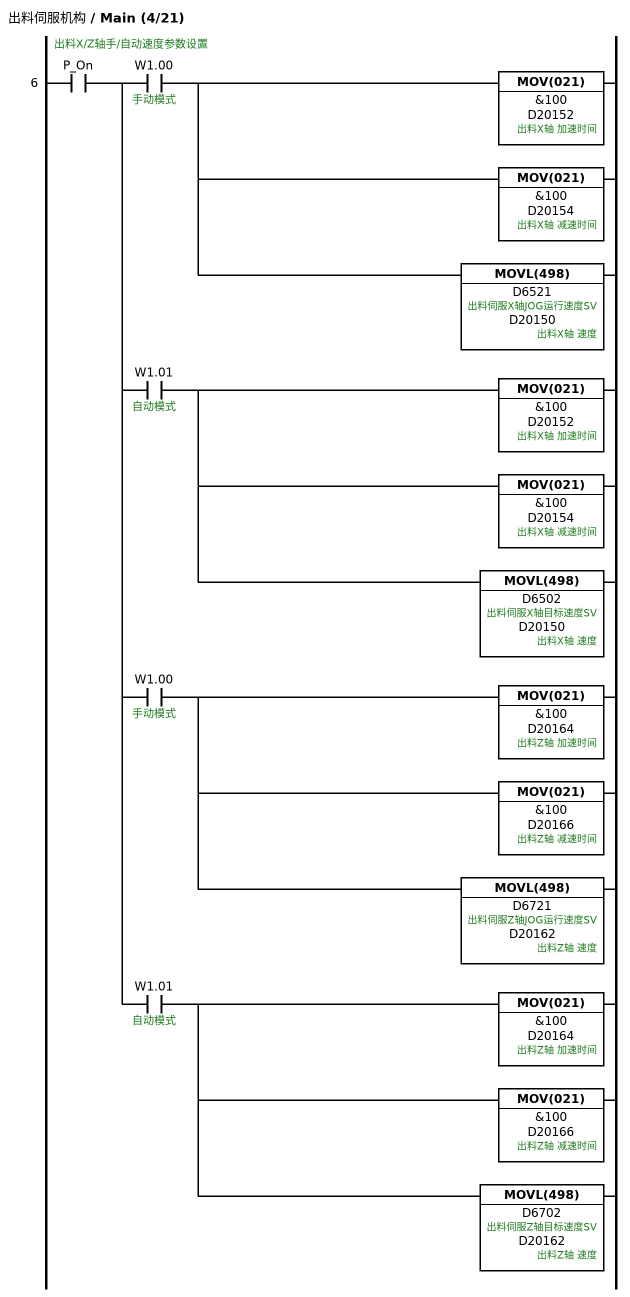
; [picture p456: 出料伺服机构 / Main, rungs 6-6]
; rung 6: 出料X/Z轴手/自动速度参数设置
LD P_On
OUT TR0
AND W1.00  ; 手动模式
MOV(021) &100 D20152  ; 出料X轴 加速时间
MOV(021) &100 D20154  ; 出料X轴 减速时间
MOVL(498) D6521 D20150  ; 出料伺服X轴JOG运行速度SV, 出料X轴 速度
LD TR0
AND W1.01  ; 自动模式
MOV(021) &100 D20152  ; 出料X轴 加速时间
MOV(021) &100 D20154  ; 出料X轴 减速时间
MOVL(498) D6502 D20150  ; 出料伺服X轴目标速度SV, 出料X轴 速度
LD TR0
AND W1.00  ; 手动模式
MOV(021) &100 D20164  ; 出料Z轴 加速时间
MOV(021) &100 D20166  ; 出料Z轴 减速时间
MOVL(498) D6721 D20162  ; 出料伺服Z轴JOG运行速度SV, 出料Z轴 速度
LD TR0
AND W1.01  ; 自动模式
MOV(021) &100 D20164  ; 出料Z轴 加速时间
MOV(021) &100 D20166  ; 出料Z轴 减速时间
MOVL(498) D6702 D20162  ; 出料伺服Z轴目标速度SV, 出料Z轴 速度

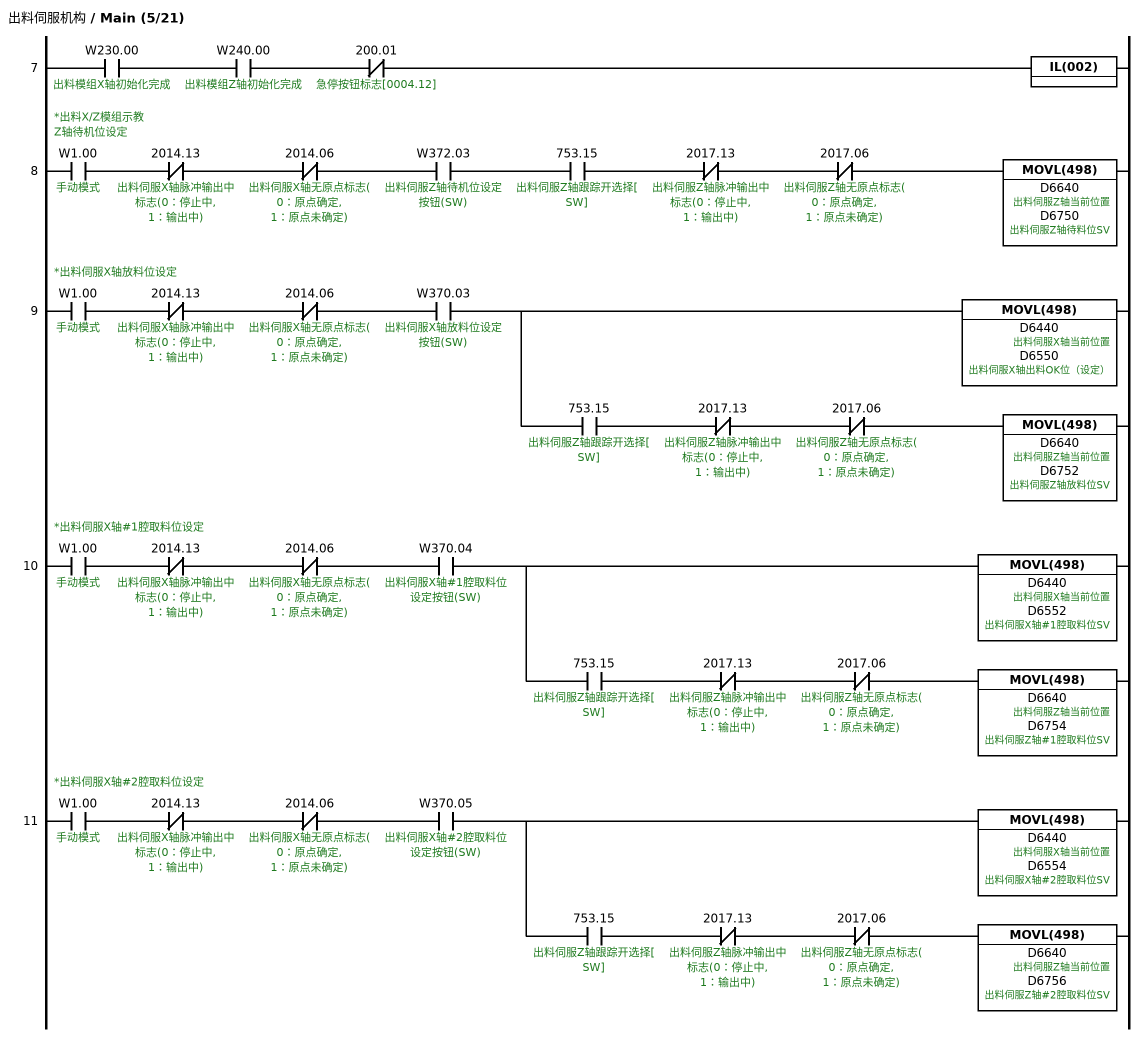
; rung 7
LD W230.00  ; 出料模组X轴初始化完成
AND W240.00  ; 出料模组Z轴初始化完成
ANDNOT 200.01  ; 急停按钮标志[0004.12]
IL(002)
; rung 8: *出料X/Z模组示教 / Z轴待机位设定
LD W1.00  ; 手动模式
ANDNOT 2014.13  ; 出料伺服X轴脉冲输出中标志(0：停止中,1：输出中)
ANDNOT 2014.06  ; 出料伺服X轴无原点标志(0：原点确定,1：原点未确定)
AND W372.03  ; 出料伺服Z轴待机位设定按钮(SW)
AND 753.15  ; 出料伺服Z轴跟踪开选择[SW]
ANDNOT 2017.13  ; 出料伺服Z轴脉冲输出中标志(0：停止中,1：输出中)
ANDNOT 2017.06  ; 出料伺服Z轴无原点标志(0：原点确定,1：原点未确定)
MOVL(498) D6640 D6750  ; 出料伺服Z轴当前位置, 出料伺服Z轴待料位SV
; rung 9: *出料伺服X轴放料位设定
LD W1.00  ; 手动模式
ANDNOT 2014.13  ; 出料伺服X轴脉冲输出中标志(0：停止中,1：输出中)
ANDNOT 2014.06  ; 出料伺服X轴无原点标志(0：原点确定,1：原点未确定)
AND W370.03  ; 出料伺服X轴放料位设定按钮(SW)
MOVL(498) D6440 D6550  ; 出料伺服X轴当前位置, 出料伺服X轴出料OK位（设定）
AND 753.15  ; 出料伺服Z轴跟踪开选择[SW]
ANDNOT 2017.13  ; 出料伺服Z轴脉冲输出中标志(0：停止中,1：输出中)
ANDNOT 2017.06  ; 出料伺服Z轴无原点标志(0：原点确定,1：原点未确定)
MOVL(498) D6640 D6752  ; 出料伺服Z轴当前位置, 出料伺服Z轴放料位SV
; rung 10: *出料伺服X轴#1腔取料位设定
LD W1.00  ; 手动模式
ANDNOT 2014.13  ; 出料伺服X轴脉冲输出中标志(0：停止中,1：输出中)
ANDNOT 2014.06  ; 出料伺服X轴无原点标志(0：原点确定,1：原点未确定)
AND W370.04  ; 出料伺服X轴#1腔取料位设定按钮(SW)
MOVL(498) D6440 D6552  ; 出料伺服X轴当前位置, 出料伺服X轴#1腔取料位SV
AND 753.15  ; 出料伺服Z轴跟踪开选择[SW]
ANDNOT 2017.13  ; 出料伺服Z轴脉冲输出中标志(0：停止中,1：输出中)
ANDNOT 2017.06  ; 出料伺服Z轴无原点标志(0：原点确定,1：原点未确定)
MOVL(498) D6640 D6754  ; 出料伺服Z轴当前位置, 出料伺服Z轴#1腔取料位SV
; rung 11: *出料伺服X轴#2腔取料位设定
LD W1.00  ; 手动模式
ANDNOT 2014.13  ; 出料伺服X轴脉冲输出中标志(0：停止中,1：输出中)
ANDNOT 2014.06  ; 出料伺服X轴无原点标志(0：原点确定,1：原点未确定)
AND W370.05  ; 出料伺服X轴#2腔取料位设定按钮(SW)
MOVL(498) D6440 D6554  ; 出料伺服X轴当前位置, 出料伺服X轴#2腔取料位SV
AND 753.15  ; 出料伺服Z轴跟踪开选择[SW]
ANDNOT 2017.13  ; 出料伺服Z轴脉冲输出中标志(0：停止中,1：输出中)
ANDNOT 2017.06  ; 出料伺服Z轴无原点标志(0：原点确定,1：原点未确定)
MOVL(498) D6640 D6756  ; 出料伺服Z轴当前位置, 出料伺服Z轴#2腔取料位SV

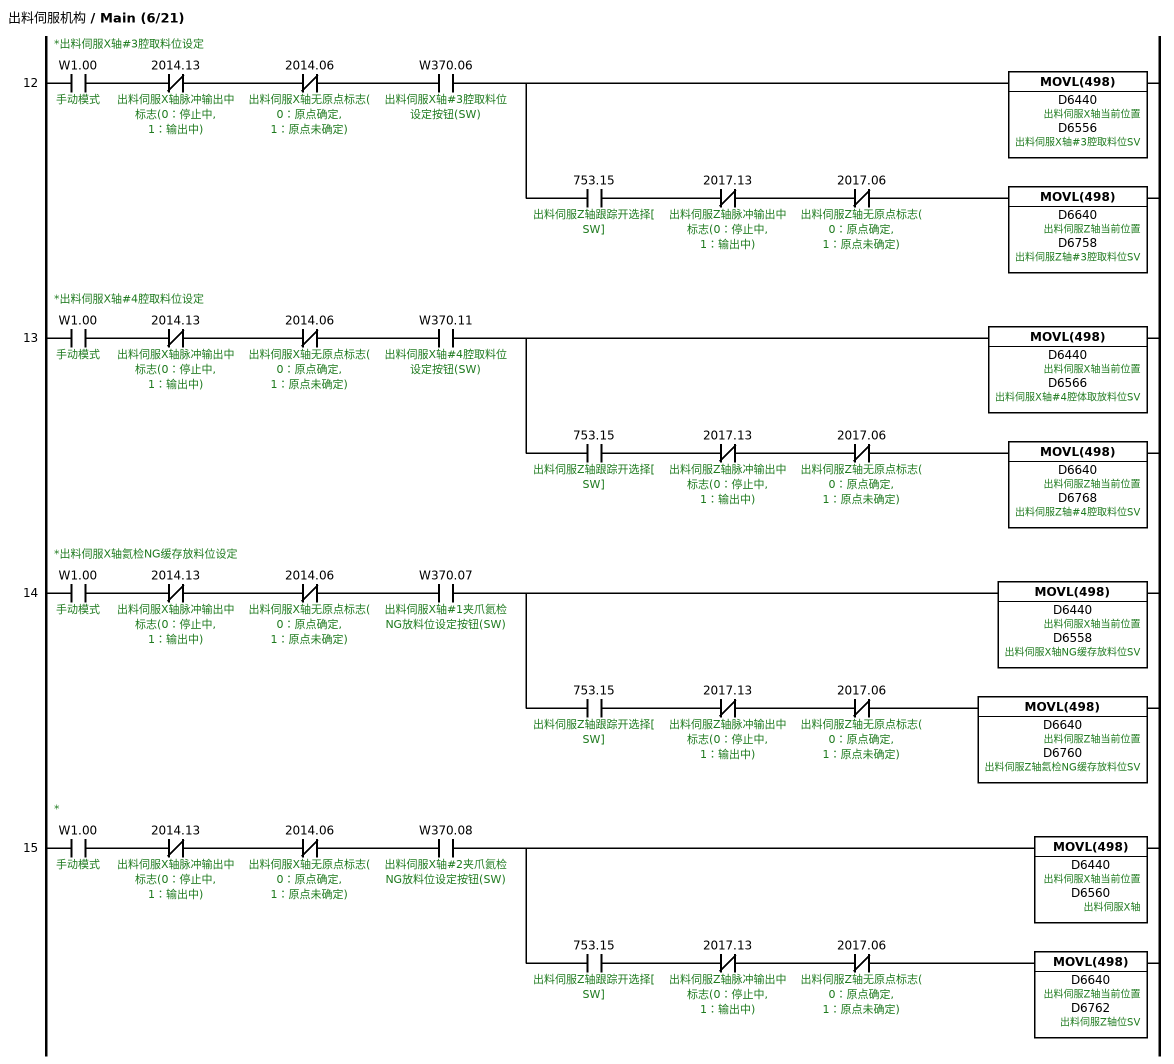
; rung 12: *出料伺服X轴#3腔取料位设定
LD W1.00  ; 手动模式
ANDNOT 2014.13  ; 出料伺服X轴脉冲输出中标志(0：停止中,1：输出中)
ANDNOT 2014.06  ; 出料伺服X轴无原点标志(0：原点确定,1：原点未确定)
AND W370.06  ; 出料伺服X轴#3腔取料位设定按钮(SW)
MOVL(498) D6440 D6556  ; 出料伺服X轴当前位置, 出料伺服X轴#3腔取料位SV
AND 753.15  ; 出料伺服Z轴跟踪开选择[SW]
ANDNOT 2017.13  ; 出料伺服Z轴脉冲输出中标志(0：停止中,1：输出中)
ANDNOT 2017.06  ; 出料伺服Z轴无原点标志(0：原点确定,1：原点未确定)
MOVL(498) D6640 D6758  ; 出料伺服Z轴当前位置, 出料伺服Z轴#3腔取料位SV
; rung 13: *出料伺服X轴#4腔取料位设定
LD W1.00  ; 手动模式
ANDNOT 2014.13  ; 出料伺服X轴脉冲输出中标志(0：停止中,1：输出中)
ANDNOT 2014.06  ; 出料伺服X轴无原点标志(0：原点确定,1：原点未确定)
AND W370.11  ; 出料伺服X轴#4腔取料位设定按钮(SW)
MOVL(498) D6440 D6566  ; 出料伺服X轴当前位置, 出料伺服X轴#4腔体取放料位SV
AND 753.15  ; 出料伺服Z轴跟踪开选择[SW]
ANDNOT 2017.13  ; 出料伺服Z轴脉冲输出中标志(0：停止中,1：输出中)
ANDNOT 2017.06  ; 出料伺服Z轴无原点标志(0：原点确定,1：原点未确定)
MOVL(498) D6640 D6768  ; 出料伺服Z轴当前位置, 出料伺服Z轴#4腔取料位SV
; rung 14: *出料伺服X轴氦检NG缓存放料位设定
LD W1.00  ; 手动模式
ANDNOT 2014.13  ; 出料伺服X轴脉冲输出中标志(0：停止中,1：输出中)
ANDNOT 2014.06  ; 出料伺服X轴无原点标志(0：原点确定,1：原点未确定)
AND W370.07  ; 出料伺服X轴#1夹爪氦检NG放料位设定按钮(SW)
MOVL(498) D6440 D6558  ; 出料伺服X轴当前位置, 出料伺服X轴NG缓存放料位SV
AND 753.15  ; 出料伺服Z轴跟踪开选择[SW]
ANDNOT 2017.13  ; 出料伺服Z轴脉冲输出中标志(0：停止中,1：输出中)
ANDNOT 2017.06  ; 出料伺服Z轴无原点标志(0：原点确定,1：原点未确定)
MOVL(498) D6640 D6760  ; 出料伺服Z轴当前位置, 出料伺服Z轴氦检NG缓存放料位SV
; rung 15: *
LD W1.00  ; 手动模式
ANDNOT 2014.13  ; 出料伺服X轴脉冲输出中标志(0：停止中,1：输出中)
ANDNOT 2014.06  ; 出料伺服X轴无原点标志(0：原点确定,1：原点未确定)
AND W370.08  ; 出料伺服X轴#2夹爪氦检NG放料位设定按钮(SW)
MOVL(498) D6440 D6560  ; 出料伺服X轴当前位置, 出料伺服X轴
AND 753.15  ; 出料伺服Z轴跟踪开选择[SW]
ANDNOT 2017.13  ; 出料伺服Z轴脉冲输出中标志(0：停止中,1：输出中)
ANDNOT 2017.06  ; 出料伺服Z轴无原点标志(0：原点确定,1：原点未确定)
MOVL(498) D6640 D6762  ; 出料伺服Z轴当前位置, 出料伺服Z轴位SV

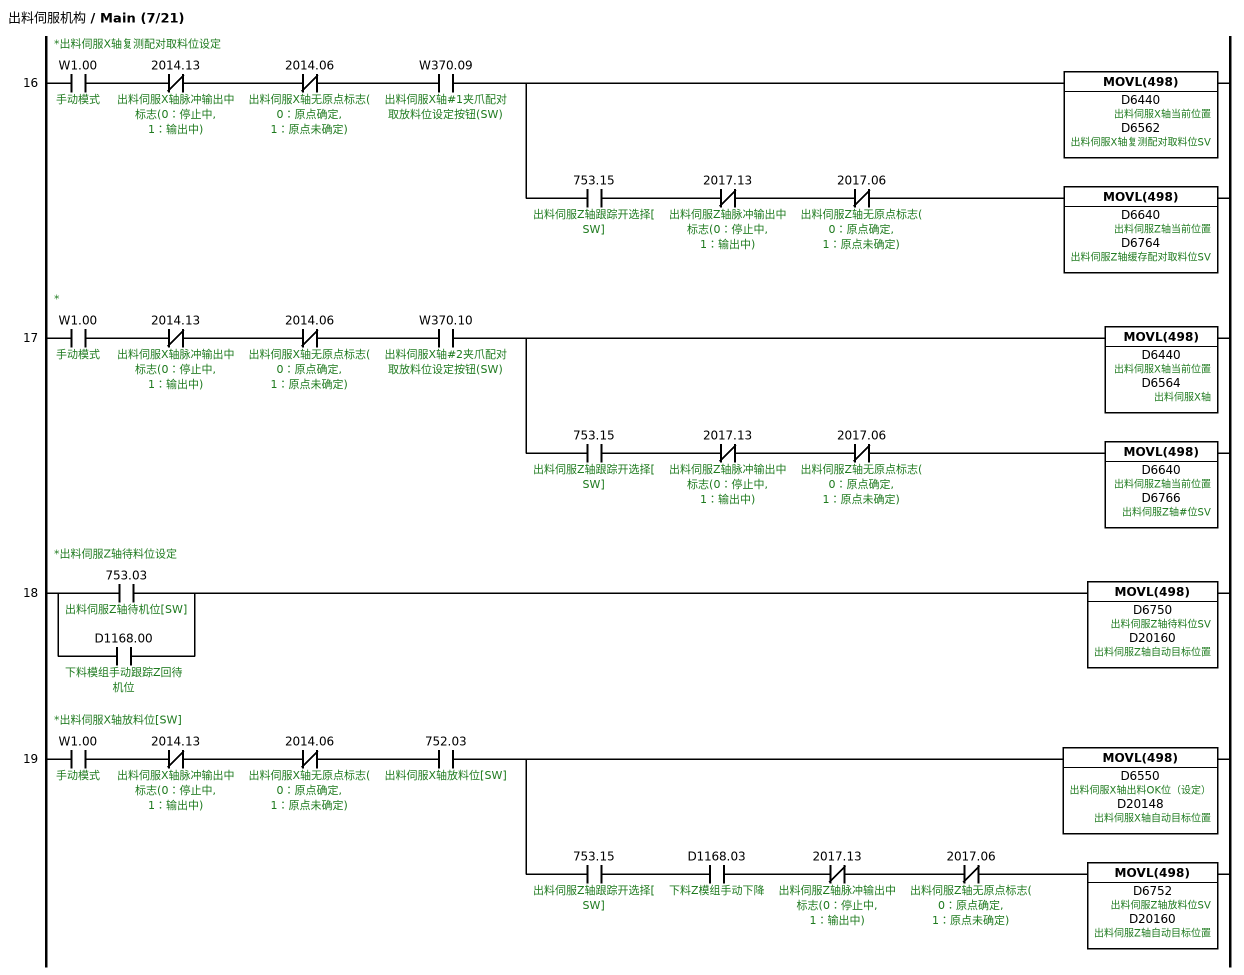
; rung 16: *出料伺服X轴复测配对取料位设定
LD W1.00  ; 手动模式
ANDNOT 2014.13  ; 出料伺服X轴脉冲输出中标志(0：停止中,1：输出中)
ANDNOT 2014.06  ; 出料伺服X轴无原点标志(0：原点确定,1：原点未确定)
AND W370.09  ; 出料伺服X轴#1夹爪配对取放料位设定按钮(SW)
MOVL(498) D6440 D6562  ; 出料伺服X轴当前位置, 出料伺服X轴复测配对取料位SV
AND 753.15  ; 出料伺服Z轴跟踪开选择[SW]
ANDNOT 2017.13  ; 出料伺服Z轴脉冲输出中标志(0：停止中,1：输出中)
ANDNOT 2017.06  ; 出料伺服Z轴无原点标志(0：原点确定,1：原点未确定)
MOVL(498) D6640 D6764  ; 出料伺服Z轴当前位置, 出料伺服Z轴缓存配对取料位SV
; rung 17: *
LD W1.00  ; 手动模式
ANDNOT 2014.13  ; 出料伺服X轴脉冲输出中标志(0：停止中,1：输出中)
ANDNOT 2014.06  ; 出料伺服X轴无原点标志(0：原点确定,1：原点未确定)
AND W370.10  ; 出料伺服X轴#2夹爪配对取放料位设定按钮(SW)
MOVL(498) D6440 D6564  ; 出料伺服X轴当前位置, 出料伺服X轴
AND 753.15  ; 出料伺服Z轴跟踪开选择[SW]
ANDNOT 2017.13  ; 出料伺服Z轴脉冲输出中标志(0：停止中,1：输出中)
ANDNOT 2017.06  ; 出料伺服Z轴无原点标志(0：原点确定,1：原点未确定)
MOVL(498) D6640 D6766  ; 出料伺服Z轴当前位置, 出料伺服Z轴#位SV
; rung 18: *出料伺服Z轴待料位设定
LD 753.03  ; 出料伺服Z轴待机位[SW]
OR D1168.00  ; 下料模组手动跟踪Z回待机位
MOVL(498) D6750 D20160  ; 出料伺服Z轴待料位SV, 出料伺服Z轴自动目标位置
; rung 19: *出料伺服X轴放料位[SW]
LD W1.00  ; 手动模式
ANDNOT 2014.13  ; 出料伺服X轴脉冲输出中标志(0：停止中,1：输出中)
ANDNOT 2014.06  ; 出料伺服X轴无原点标志(0：原点确定,1：原点未确定)
AND 752.03  ; 出料伺服X轴放料位[SW]
MOVL(498) D6550 D20148  ; 出料伺服X轴出料OK位（设定）, 出料伺服X轴自动目标位置
AND 753.15  ; 出料伺服Z轴跟踪开选择[SW]
AND D1168.03  ; 下料Z模组手动下降
ANDNOT 2017.13  ; 出料伺服Z轴脉冲输出中标志(0：停止中,1：输出中)
ANDNOT 2017.06  ; 出料伺服Z轴无原点标志(0：原点确定,1：原点未确定)
MOVL(498) D6752 D20160  ; 出料伺服Z轴放料位SV, 出料伺服Z轴自动目标位置

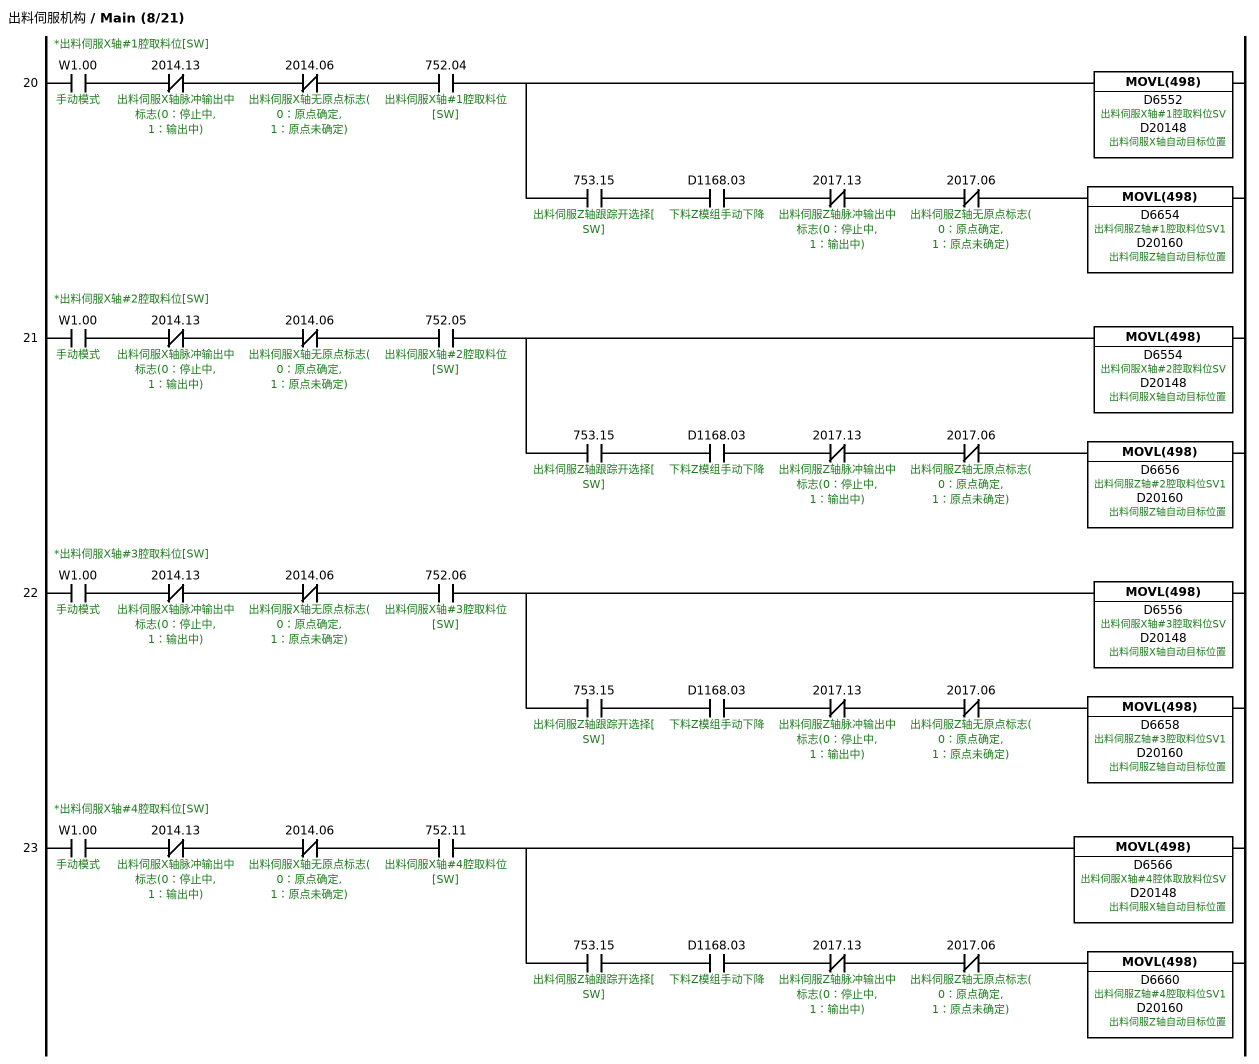
; rung 20: *出料伺服X轴#1腔取料位[SW]
LD W1.00  ; 手动模式
ANDNOT 2014.13  ; 出料伺服X轴脉冲输出中标志(0：停止中,1：输出中)
ANDNOT 2014.06  ; 出料伺服X轴无原点标志(0：原点确定,1：原点未确定)
AND 752.04  ; 出料伺服X轴#1腔取料位[SW]
MOVL(498) D6552 D20148  ; 出料伺服X轴#1腔取料位SV, 出料伺服X轴自动目标位置
AND 753.15  ; 出料伺服Z轴跟踪开选择[SW]
AND D1168.03  ; 下料Z模组手动下降
ANDNOT 2017.13  ; 出料伺服Z轴脉冲输出中标志(0：停止中,1：输出中)
ANDNOT 2017.06  ; 出料伺服Z轴无原点标志(0：原点确定,1：原点未确定)
MOVL(498) D6654 D20160  ; 出料伺服Z轴#1腔取料位SV1, 出料伺服Z轴自动目标位置
; rung 21: *出料伺服X轴#2腔取料位[SW]
LD W1.00  ; 手动模式
ANDNOT 2014.13  ; 出料伺服X轴脉冲输出中标志(0：停止中,1：输出中)
ANDNOT 2014.06  ; 出料伺服X轴无原点标志(0：原点确定,1：原点未确定)
AND 752.05  ; 出料伺服X轴#2腔取料位[SW]
MOVL(498) D6554 D20148  ; 出料伺服X轴#2腔取料位SV, 出料伺服X轴自动目标位置
AND 753.15  ; 出料伺服Z轴跟踪开选择[SW]
AND D1168.03  ; 下料Z模组手动下降
ANDNOT 2017.13  ; 出料伺服Z轴脉冲输出中标志(0：停止中,1：输出中)
ANDNOT 2017.06  ; 出料伺服Z轴无原点标志(0：原点确定,1：原点未确定)
MOVL(498) D6656 D20160  ; 出料伺服Z轴#2腔取料位SV1, 出料伺服Z轴自动目标位置
; rung 22: *出料伺服X轴#3腔取料位[SW]
LD W1.00  ; 手动模式
ANDNOT 2014.13  ; 出料伺服X轴脉冲输出中标志(0：停止中,1：输出中)
ANDNOT 2014.06  ; 出料伺服X轴无原点标志(0：原点确定,1：原点未确定)
AND 752.06  ; 出料伺服X轴#3腔取料位[SW]
MOVL(498) D6556 D20148  ; 出料伺服X轴#3腔取料位SV, 出料伺服X轴自动目标位置
AND 753.15  ; 出料伺服Z轴跟踪开选择[SW]
AND D1168.03  ; 下料Z模组手动下降
ANDNOT 2017.13  ; 出料伺服Z轴脉冲输出中标志(0：停止中,1：输出中)
ANDNOT 2017.06  ; 出料伺服Z轴无原点标志(0：原点确定,1：原点未确定)
MOVL(498) D6658 D20160  ; 出料伺服Z轴#3腔取料位SV1, 出料伺服Z轴自动目标位置
; rung 23: *出料伺服X轴#4腔取料位[SW]
LD W1.00  ; 手动模式
ANDNOT 2014.13  ; 出料伺服X轴脉冲输出中标志(0：停止中,1：输出中)
ANDNOT 2014.06  ; 出料伺服X轴无原点标志(0：原点确定,1：原点未确定)
AND 752.11  ; 出料伺服X轴#4腔取料位[SW]
MOVL(498) D6566 D20148  ; 出料伺服X轴#4腔体取放料位SV, 出料伺服X轴自动目标位置
AND 753.15  ; 出料伺服Z轴跟踪开选择[SW]
AND D1168.03  ; 下料Z模组手动下降
ANDNOT 2017.13  ; 出料伺服Z轴脉冲输出中标志(0：停止中,1：输出中)
ANDNOT 2017.06  ; 出料伺服Z轴无原点标志(0：原点确定,1：原点未确定)
MOVL(498) D6660 D20160  ; 出料伺服Z轴#4腔取料位SV1, 出料伺服Z轴自动目标位置

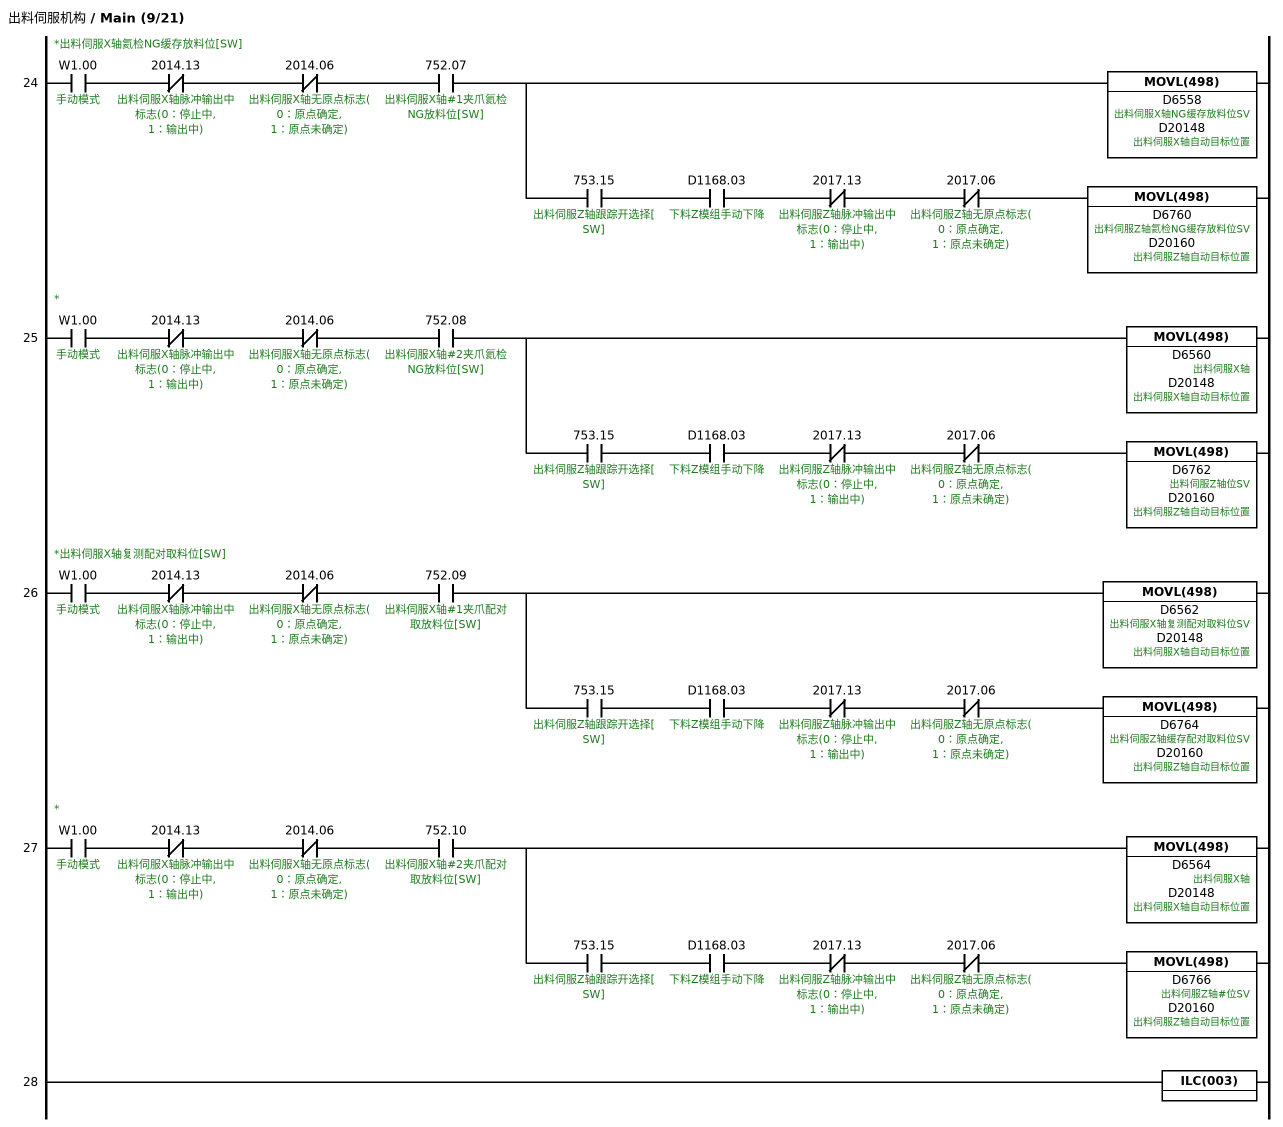
; rung 24: *出料伺服X轴氦检NG缓存放料位[SW]
LD W1.00  ; 手动模式
ANDNOT 2014.13  ; 出料伺服X轴脉冲输出中标志(0：停止中,1：输出中)
ANDNOT 2014.06  ; 出料伺服X轴无原点标志(0：原点确定,1：原点未确定)
AND 752.07  ; 出料伺服X轴#1夹爪氦检NG放料位[SW]
MOVL(498) D6558 D20148  ; 出料伺服X轴NG缓存放料位SV, 出料伺服X轴自动目标位置
AND 753.15  ; 出料伺服Z轴跟踪开选择[SW]
AND D1168.03  ; 下料Z模组手动下降
ANDNOT 2017.13  ; 出料伺服Z轴脉冲输出中标志(0：停止中,1：输出中)
ANDNOT 2017.06  ; 出料伺服Z轴无原点标志(0：原点确定,1：原点未确定)
MOVL(498) D6760 D20160  ; 出料伺服Z轴氦检NG缓存放料位SV, 出料伺服Z轴自动目标位置
; rung 25: *
LD W1.00  ; 手动模式
ANDNOT 2014.13  ; 出料伺服X轴脉冲输出中标志(0：停止中,1：输出中)
ANDNOT 2014.06  ; 出料伺服X轴无原点标志(0：原点确定,1：原点未确定)
AND 752.08  ; 出料伺服X轴#2夹爪氦检NG放料位[SW]
MOVL(498) D6560 D20148  ; 出料伺服X轴, 出料伺服X轴自动目标位置
AND 753.15  ; 出料伺服Z轴跟踪开选择[SW]
AND D1168.03  ; 下料Z模组手动下降
ANDNOT 2017.13  ; 出料伺服Z轴脉冲输出中标志(0：停止中,1：输出中)
ANDNOT 2017.06  ; 出料伺服Z轴无原点标志(0：原点确定,1：原点未确定)
MOVL(498) D6762 D20160  ; 出料伺服Z轴位SV, 出料伺服Z轴自动目标位置
; rung 26: *出料伺服X轴复测配对取料位[SW]
LD W1.00  ; 手动模式
ANDNOT 2014.13  ; 出料伺服X轴脉冲输出中标志(0：停止中,1：输出中)
ANDNOT 2014.06  ; 出料伺服X轴无原点标志(0：原点确定,1：原点未确定)
AND 752.09  ; 出料伺服X轴#1夹爪配对取放料位[SW]
MOVL(498) D6562 D20148  ; 出料伺服X轴复测配对取料位SV, 出料伺服X轴自动目标位置
AND 753.15  ; 出料伺服Z轴跟踪开选择[SW]
AND D1168.03  ; 下料Z模组手动下降
ANDNOT 2017.13  ; 出料伺服Z轴脉冲输出中标志(0：停止中,1：输出中)
ANDNOT 2017.06  ; 出料伺服Z轴无原点标志(0：原点确定,1：原点未确定)
MOVL(498) D6764 D20160  ; 出料伺服Z轴缓存配对取料位SV, 出料伺服Z轴自动目标位置
; rung 27: *
LD W1.00  ; 手动模式
ANDNOT 2014.13  ; 出料伺服X轴脉冲输出中标志(0：停止中,1：输出中)
ANDNOT 2014.06  ; 出料伺服X轴无原点标志(0：原点确定,1：原点未确定)
AND 752.10  ; 出料伺服X轴#2夹爪配对取放料位[SW]
MOVL(498) D6564 D20148  ; 出料伺服X轴, 出料伺服X轴自动目标位置
AND 753.15  ; 出料伺服Z轴跟踪开选择[SW]
AND D1168.03  ; 下料Z模组手动下降
ANDNOT 2017.13  ; 出料伺服Z轴脉冲输出中标志(0：停止中,1：输出中)
ANDNOT 2017.06  ; 出料伺服Z轴无原点标志(0：原点确定,1：原点未确定)
MOVL(498) D6766 D20160  ; 出料伺服Z轴#位SV, 出料伺服Z轴自动目标位置
; rung 28
ILC(003)

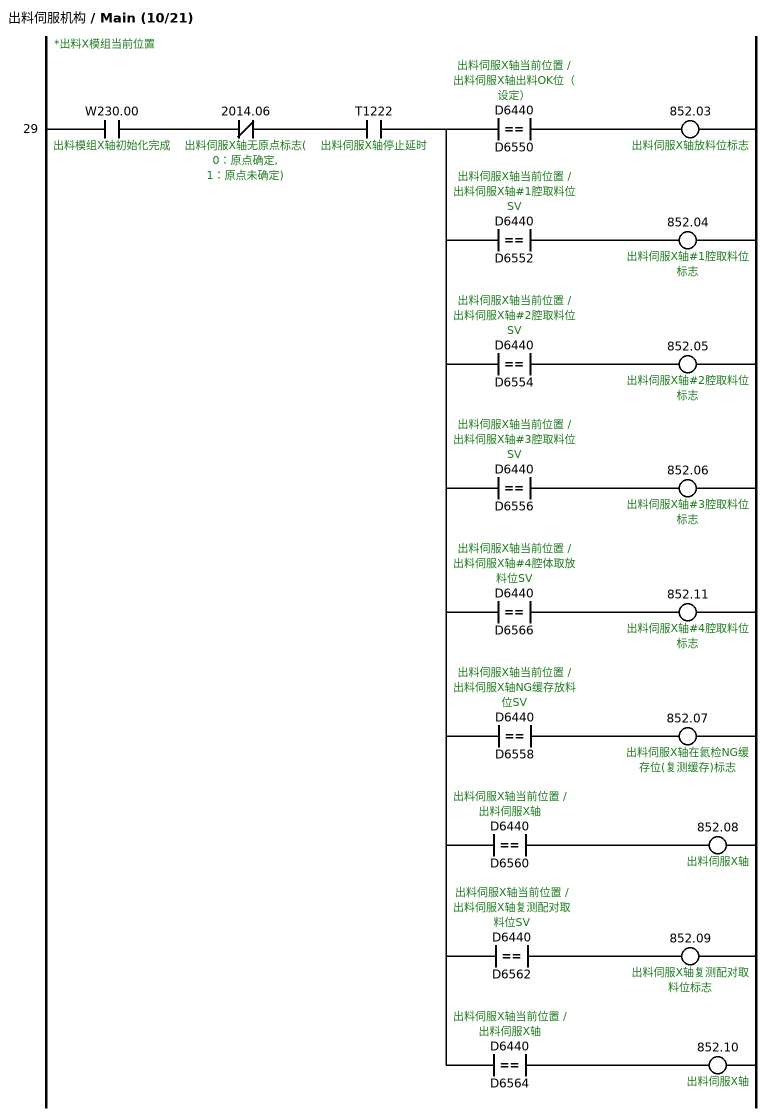
; rung 29: *出料X模组当前位置
LD W230.00  ; 出料模组X轴初始化完成
ANDNOT 2014.06  ; 出料伺服X轴无原点标志(0：原点确定,1：原点未确定)
AND T1222  ; 出料伺服X轴停止延时
OUT TR0
AND=SL(303) D6440 D6550  ; 出料伺服X轴当前位置, 出料伺服X轴出料OK位（设定）
OUT 852.03  ; 出料伺服X轴放料位标志
LD TR0
AND=SL(303) D6440 D6552  ; 出料伺服X轴当前位置, 出料伺服X轴#1腔取料位SV
OUT 852.04  ; 出料伺服X轴#1腔取料位标志
LD TR0
AND=SL(303) D6440 D6554  ; 出料伺服X轴当前位置, 出料伺服X轴#2腔取料位SV
OUT 852.05  ; 出料伺服X轴#2腔取料位标志
LD TR0
AND=SL(303) D6440 D6556  ; 出料伺服X轴当前位置, 出料伺服X轴#3腔取料位SV
OUT 852.06  ; 出料伺服X轴#3腔取料位标志
LD TR0
AND=SL(303) D6440 D6566  ; 出料伺服X轴当前位置, 出料伺服X轴#4腔体取放料位SV
OUT 852.11  ; 出料伺服X轴#4腔取料位标志
LD TR0
AND=SL(303) D6440 D6558  ; 出料伺服X轴当前位置, 出料伺服X轴NG缓存放料位SV
OUT 852.07  ; 出料伺服X轴在氦检NG缓存位(复测缓存)标志
LD TR0
AND=SL(303) D6440 D6560  ; 出料伺服X轴当前位置, 出料伺服X轴
OUT 852.08  ; 出料伺服X轴
LD TR0
AND=SL(303) D6440 D6562  ; 出料伺服X轴当前位置, 出料伺服X轴复测配对取料位SV
OUT 852.09  ; 出料伺服X轴复测配对取料位标志
LD TR0
AND=SL(303) D6440 D6564  ; 出料伺服X轴当前位置, 出料伺服X轴
OUT 852.10  ; 出料伺服X轴

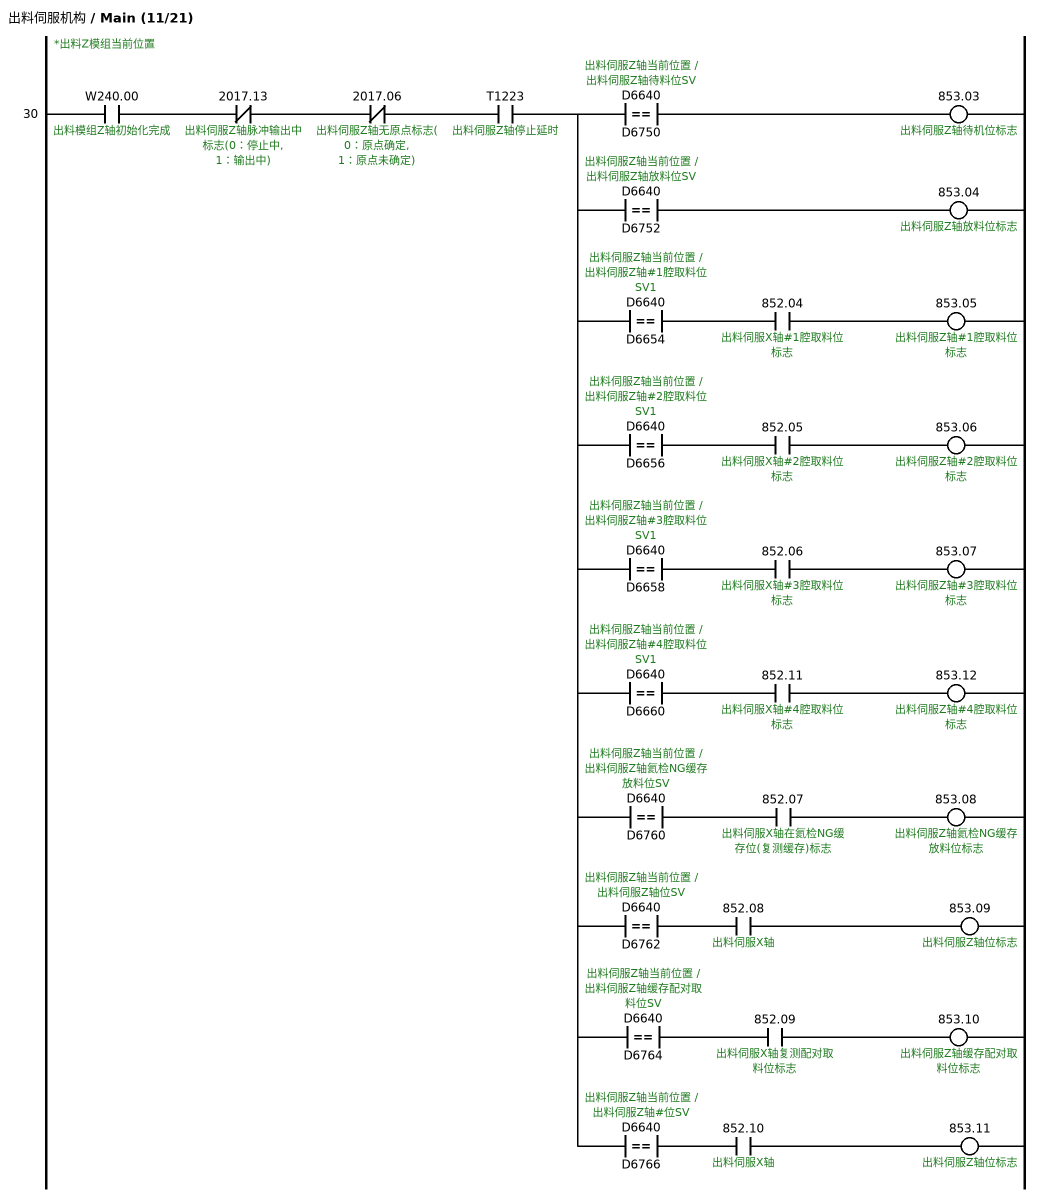
; rung 30: *出料Z模组当前位置
LD W240.00  ; 出料模组Z轴初始化完成
ANDNOT 2017.13  ; 出料伺服Z轴脉冲输出中标志(0：停止中,1：输出中)
ANDNOT 2017.06  ; 出料伺服Z轴无原点标志(0：原点确定,1：原点未确定)
AND T1223  ; 出料伺服Z轴停止延时
OUT TR0
AND=SL(303) D6640 D6750  ; 出料伺服Z轴当前位置, 出料伺服Z轴待料位SV
OUT 853.03  ; 出料伺服Z轴待机位标志
LD TR0
AND=SL(303) D6640 D6752  ; 出料伺服Z轴当前位置, 出料伺服Z轴放料位SV
OUT 853.04  ; 出料伺服Z轴放料位标志
LD TR0
AND=SL(303) D6640 D6654  ; 出料伺服Z轴当前位置, 出料伺服Z轴#1腔取料位SV1
AND 852.04  ; 出料伺服X轴#1腔取料位标志
OUT 853.05  ; 出料伺服Z轴#1腔取料位标志
LD TR0
AND=SL(303) D6640 D6656  ; 出料伺服Z轴当前位置, 出料伺服Z轴#2腔取料位SV1
AND 852.05  ; 出料伺服X轴#2腔取料位标志
OUT 853.06  ; 出料伺服Z轴#2腔取料位标志
LD TR0
AND=SL(303) D6640 D6658  ; 出料伺服Z轴当前位置, 出料伺服Z轴#3腔取料位SV1
AND 852.06  ; 出料伺服X轴#3腔取料位标志
OUT 853.07  ; 出料伺服Z轴#3腔取料位标志
LD TR0
AND=SL(303) D6640 D6660  ; 出料伺服Z轴当前位置, 出料伺服Z轴#4腔取料位SV1
AND 852.11  ; 出料伺服X轴#4腔取料位标志
OUT 853.12  ; 出料伺服Z轴#4腔取料位标志
LD TR0
AND=SL(303) D6640 D6760  ; 出料伺服Z轴当前位置, 出料伺服Z轴氦检NG缓存放料位SV
AND 852.07  ; 出料伺服X轴在氦检NG缓存位(复测缓存)标志
OUT 853.08  ; 出料伺服Z轴氦检NG缓存放料位标志
LD TR0
AND=SL(303) D6640 D6762  ; 出料伺服Z轴当前位置, 出料伺服Z轴位SV
AND 852.08  ; 出料伺服X轴
OUT 853.09  ; 出料伺服Z轴位标志
LD TR0
AND=SL(303) D6640 D6764  ; 出料伺服Z轴当前位置, 出料伺服Z轴缓存配对取料位SV
AND 852.09  ; 出料伺服X轴复测配对取料位标志
OUT 853.10  ; 出料伺服Z轴缓存配对取料位标志
LD TR0
AND=SL(303) D6640 D6766  ; 出料伺服Z轴当前位置, 出料伺服Z轴#位SV
AND 852.10  ; 出料伺服X轴
OUT 853.11  ; 出料伺服Z轴位标志

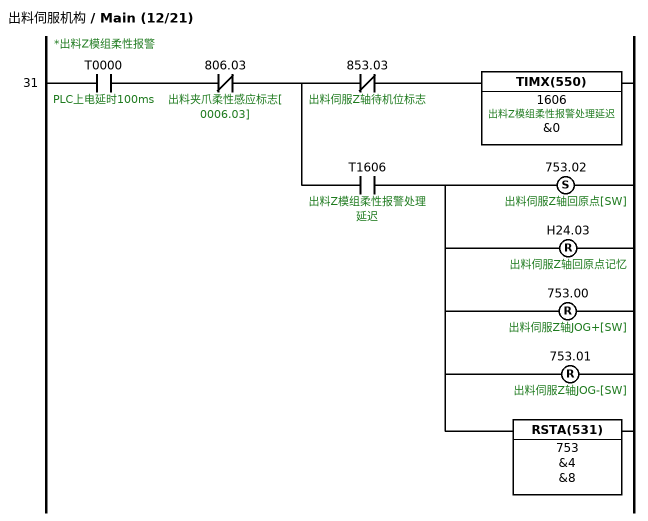
; rung 31: *出料Z模组柔性报警
LD T0000  ; PLC上电延时100ms
ANDNOT 806.03  ; 出料夹爪柔性感应标志[0006.03]
OUT TR0
ANDNOT 853.03  ; 出料伺服Z轴待机位标志
TIMX(550) 1606 &0  ; 出料Z模组柔性报警处理延迟
LD TR0
AND T1606  ; 出料Z模组柔性报警处理延迟
SET 753.02  ; 出料伺服Z轴回原点[SW]
RSET H24.03  ; 出料伺服Z轴回原点记忆
RSET 753.00  ; 出料伺服Z轴JOG+[SW]
RSET 753.01  ; 出料伺服Z轴JOG-[SW]
RSTA(531) 753 &4 &8

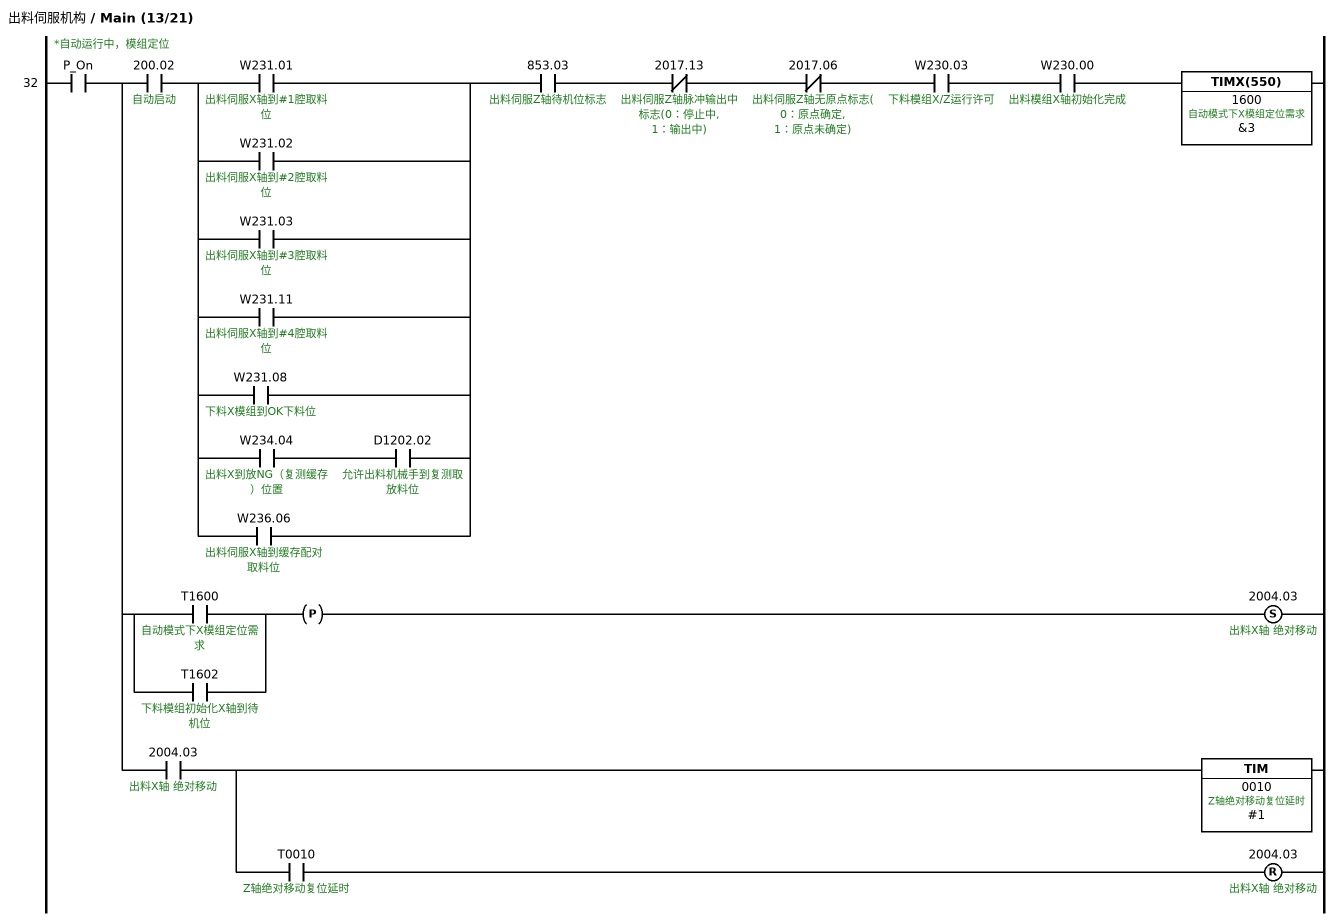
; rung 32: *自动运行中，模组定位
LD P_On
OUT TR0
AND 200.02  ; 自动启动
LD W231.01  ; 出料伺服X轴到#1腔取料位
OR W231.02  ; 出料伺服X轴到#2腔取料位
OR W231.03  ; 出料伺服X轴到#3腔取料位
OR W231.11  ; 出料伺服X轴到#4腔取料位
OR W231.08  ; 下料X模组到OK下料位
LD W234.04  ; 出料X到放NG（复测缓存）位置
AND D1202.02  ; 允许出料机械手到复测取放料位
ORLD
OR W236.06  ; 出料伺服X轴到缓存配对取料位
ANDLD
AND 853.03  ; 出料伺服Z轴待机位标志
ANDNOT 2017.13  ; 出料伺服Z轴脉冲输出中标志(0：停止中,1：输出中)
ANDNOT 2017.06  ; 出料伺服Z轴无原点标志(0：原点确定,1：原点未确定)
AND W230.03  ; 下料模组X/Z运行许可
AND W230.00  ; 出料模组X轴初始化完成
TIMX(550) 1600 &3  ; 自动模式下X模组定位需求
LD TR0
LD T1600  ; 自动模式下X模组定位需求
OR T1602  ; 下料模组初始化X轴到待机位
ANDLD
UP(521)
SET 2004.03  ; 出料X轴 绝对移动
LD TR0
AND 2004.03  ; 出料X轴 绝对移动
TIM 0010 #1  ; Z轴绝对移动复位延时
AND T0010  ; Z轴绝对移动复位延时
RSET 2004.03  ; 出料X轴 绝对移动

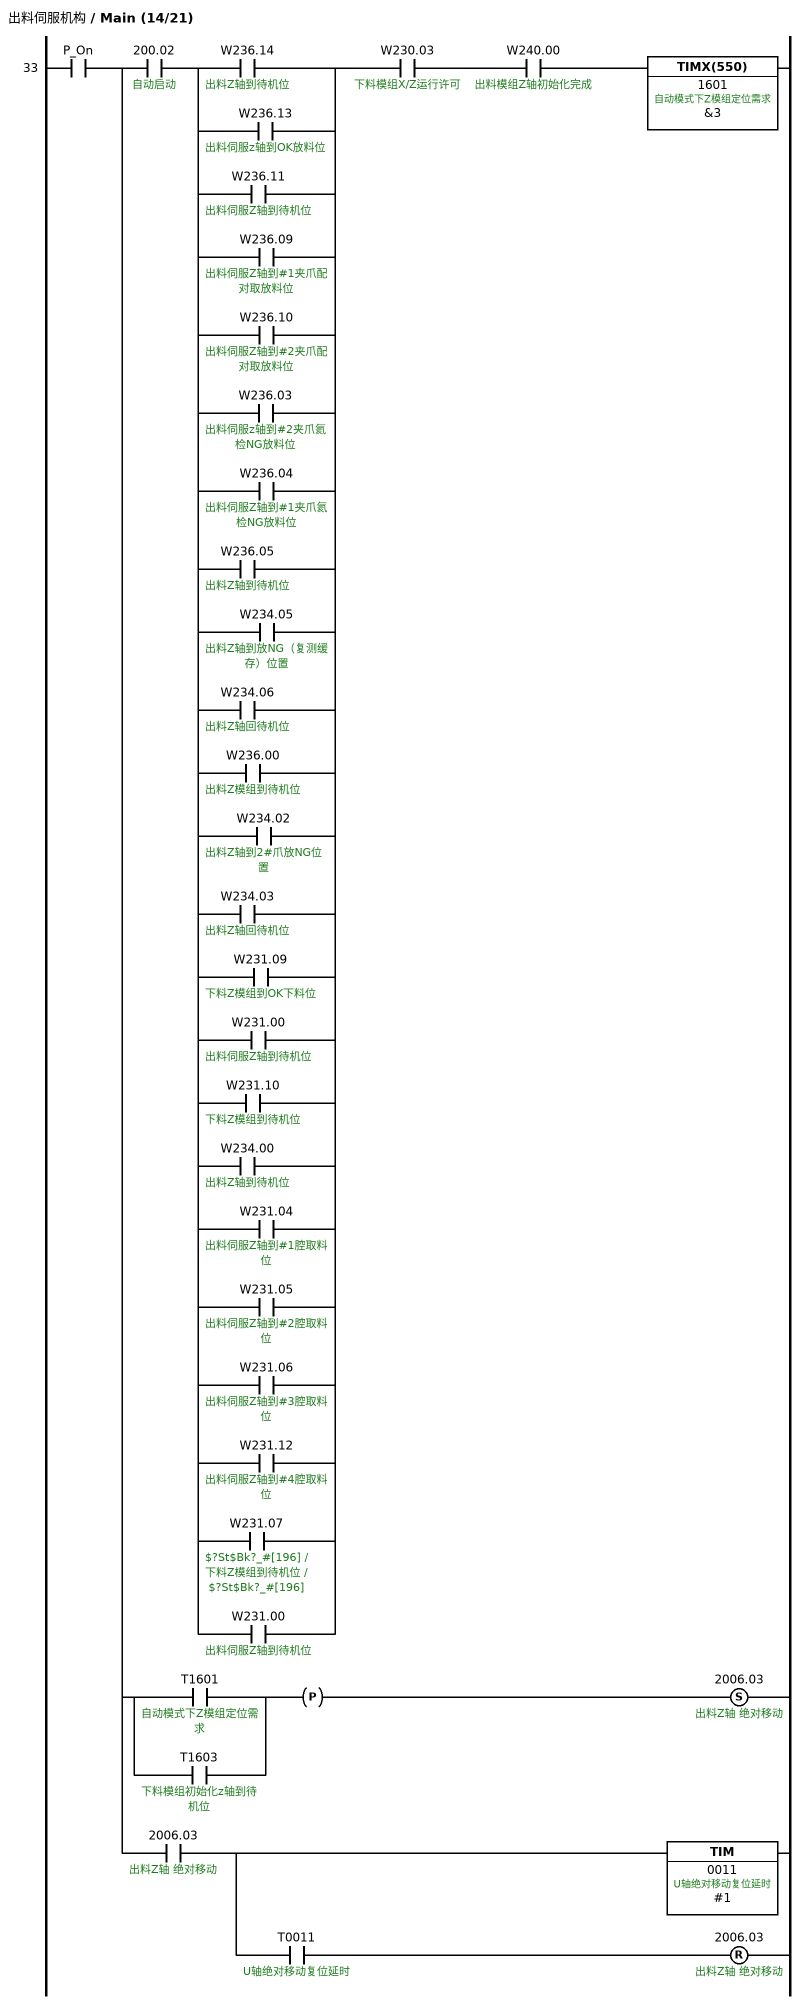
; rung 33
LD P_On
OUT TR0
AND 200.02  ; 自动启动
LD W236.14  ; 出料Z轴到待机位
OR W236.13  ; 出料伺服z轴到OK放料位
OR W236.11  ; 出料伺服Z轴到待机位
OR W236.09  ; 出料伺服Z轴到#1夹爪配对取放料位
OR W236.10  ; 出料伺服Z轴到#2夹爪配对取放料位
OR W236.03  ; 出料伺服z轴到#2夹爪氦检NG放料位
OR W236.04  ; 出料伺服Z轴到#1夹爪氦检NG放料位
OR W236.05  ; 出料Z轴到待机位
OR W234.05  ; 出料Z轴到放NG（复测缓存）位置
OR W234.06  ; 出料Z轴回待机位
OR W236.00  ; 出料Z模组到待机位
OR W234.02  ; 出料Z轴到2#爪放NG位置
OR W234.03  ; 出料Z轴回待机位
OR W231.09  ; 下料Z模组到OK下料位
OR W231.00  ; 出料伺服Z轴到待机位
OR W231.10  ; 下料Z模组到待机位
OR W234.00  ; 出料Z轴到待机位
OR W231.04  ; 出料伺服Z轴到#1腔取料位
OR W231.05  ; 出料伺服Z轴到#2腔取料位
OR W231.06  ; 出料伺服Z轴到#3腔取料位
OR W231.12  ; 出料伺服Z轴到#4腔取料位
OR W231.07  ; $?St$Bk?_#[196] / 下料Z模组到待机位 / $?St$Bk?_#[196]
OR W231.00  ; 出料伺服Z轴到待机位
ANDLD
AND W230.03  ; 下料模组X/Z运行许可
AND W240.00  ; 出料模组Z轴初始化完成
TIMX(550) 1601 &3  ; 自动模式下Z模组定位需求
LD TR0
LD T1601  ; 自动模式下Z模组定位需求
OR T1603  ; 下料模组初始化z轴到待机位
ANDLD
UP(521)
SET 2006.03  ; 出料Z轴 绝对移动
LD TR0
AND 2006.03  ; 出料Z轴 绝对移动
TIM 0011 #1  ; U轴绝对移动复位延时
AND T0011  ; U轴绝对移动复位延时
RSET 2006.03  ; 出料Z轴 绝对移动

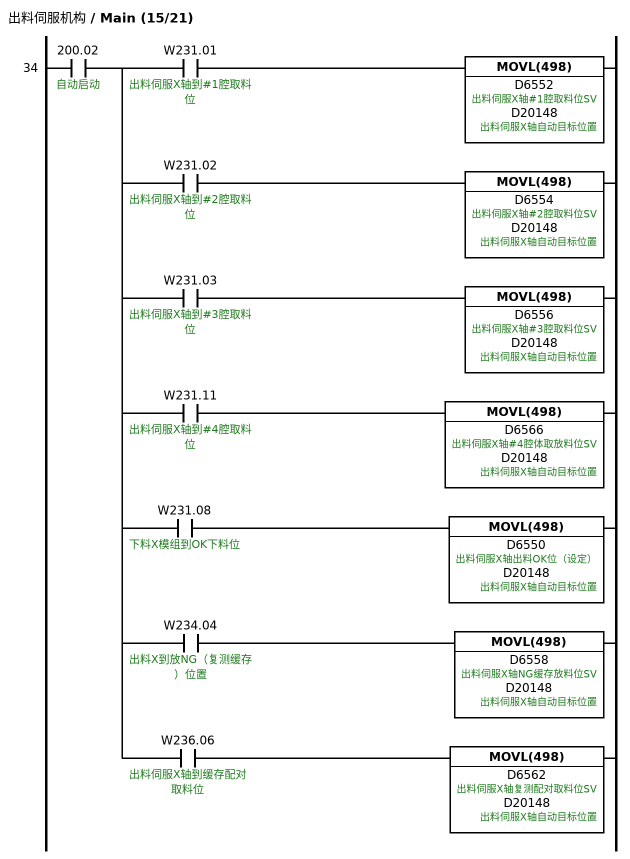
; rung 34
LD 200.02  ; 自动启动
OUT TR0
AND W231.01  ; 出料伺服X轴到#1腔取料位
MOVL(498) D6552 D20148  ; 出料伺服X轴#1腔取料位SV, 出料伺服X轴自动目标位置
LD TR0
AND W231.02  ; 出料伺服X轴到#2腔取料位
MOVL(498) D6554 D20148  ; 出料伺服X轴#2腔取料位SV, 出料伺服X轴自动目标位置
LD TR0
AND W231.03  ; 出料伺服X轴到#3腔取料位
MOVL(498) D6556 D20148  ; 出料伺服X轴#3腔取料位SV, 出料伺服X轴自动目标位置
LD TR0
AND W231.11  ; 出料伺服X轴到#4腔取料位
MOVL(498) D6566 D20148  ; 出料伺服X轴#4腔体取放料位SV, 出料伺服X轴自动目标位置
LD TR0
AND W231.08  ; 下料X模组到OK下料位
MOVL(498) D6550 D20148  ; 出料伺服X轴出料OK位（设定）, 出料伺服X轴自动目标位置
LD TR0
AND W234.04  ; 出料X到放NG（复测缓存）位置
MOVL(498) D6558 D20148  ; 出料伺服X轴NG缓存放料位SV, 出料伺服X轴自动目标位置
LD TR0
AND W236.06  ; 出料伺服X轴到缓存配对取料位
MOVL(498) D6562 D20148  ; 出料伺服X轴复测配对取料位SV, 出料伺服X轴自动目标位置

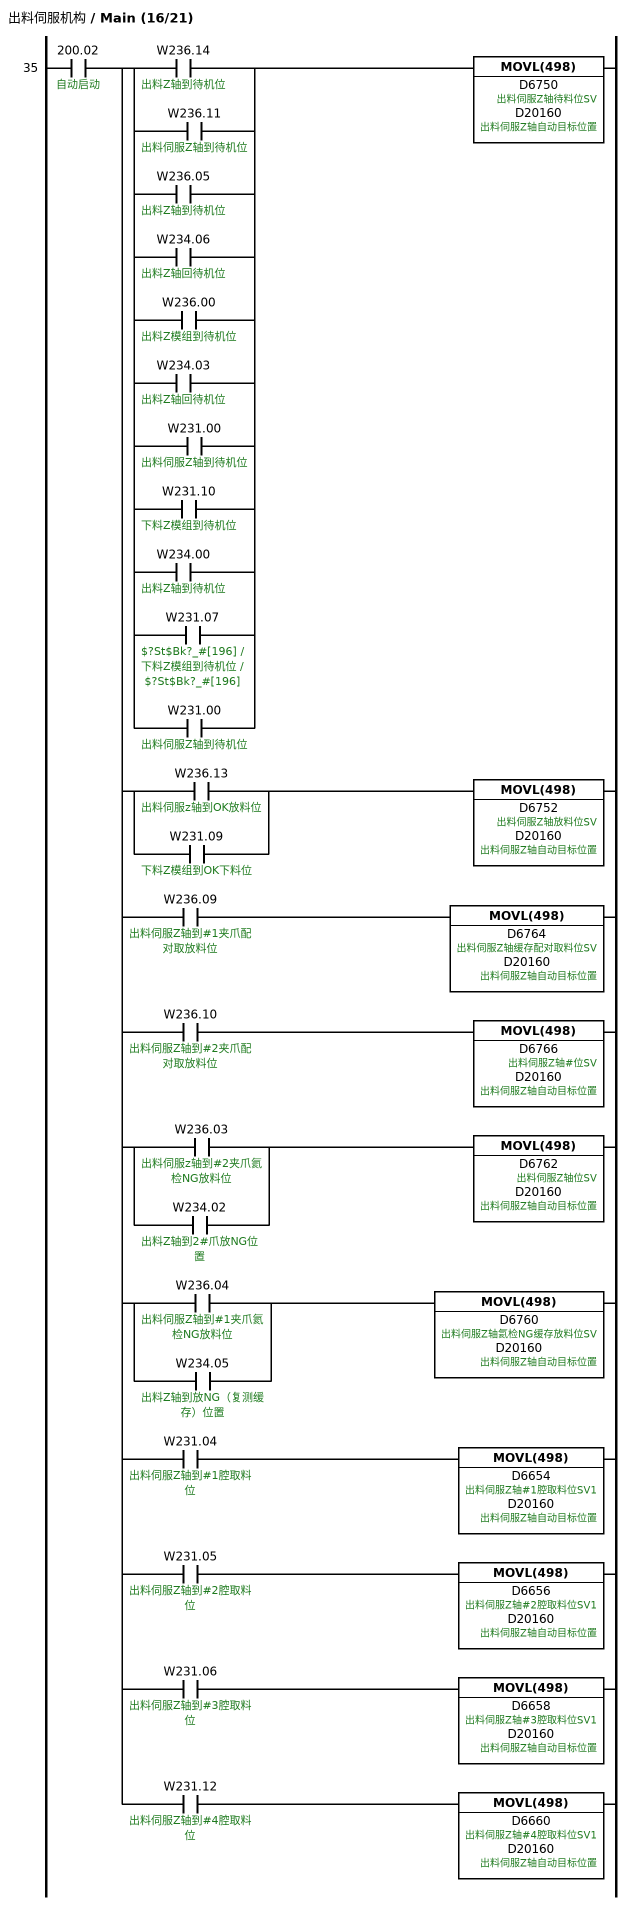
; rung 35
LD 200.02  ; 自动启动
OUT TR0
LD W236.14  ; 出料Z轴到待机位
OR W236.11  ; 出料伺服Z轴到待机位
OR W236.05  ; 出料Z轴到待机位
OR W234.06  ; 出料Z轴回待机位
OR W236.00  ; 出料Z模组到待机位
OR W234.03  ; 出料Z轴回待机位
OR W231.00  ; 出料伺服Z轴到待机位
OR W231.10  ; 下料Z模组到待机位
OR W234.00  ; 出料Z轴到待机位
OR W231.07  ; $?St$Bk?_#[196] / 下料Z模组到待机位 / $?St$Bk?_#[196]
OR W231.00  ; 出料伺服Z轴到待机位
ANDLD
MOVL(498) D6750 D20160  ; 出料伺服Z轴待料位SV, 出料伺服Z轴自动目标位置
LD TR0
LD W236.13  ; 出料伺服z轴到OK放料位
OR W231.09  ; 下料Z模组到OK下料位
ANDLD
MOVL(498) D6752 D20160  ; 出料伺服Z轴放料位SV, 出料伺服Z轴自动目标位置
LD TR0
AND W236.09  ; 出料伺服Z轴到#1夹爪配对取放料位
MOVL(498) D6764 D20160  ; 出料伺服Z轴缓存配对取料位SV, 出料伺服Z轴自动目标位置
LD TR0
AND W236.10  ; 出料伺服Z轴到#2夹爪配对取放料位
MOVL(498) D6766 D20160  ; 出料伺服Z轴#位SV, 出料伺服Z轴自动目标位置
LD TR0
LD W236.03  ; 出料伺服z轴到#2夹爪氦检NG放料位
OR W234.02  ; 出料Z轴到2#爪放NG位置
ANDLD
MOVL(498) D6762 D20160  ; 出料伺服Z轴位SV, 出料伺服Z轴自动目标位置
LD TR0
LD W236.04  ; 出料伺服Z轴到#1夹爪氦检NG放料位
OR W234.05  ; 出料Z轴到放NG（复测缓存）位置
ANDLD
MOVL(498) D6760 D20160  ; 出料伺服Z轴氦检NG缓存放料位SV, 出料伺服Z轴自动目标位置
LD TR0
AND W231.04  ; 出料伺服Z轴到#1腔取料位
MOVL(498) D6654 D20160  ; 出料伺服Z轴#1腔取料位SV1, 出料伺服Z轴自动目标位置
LD TR0
AND W231.05  ; 出料伺服Z轴到#2腔取料位
MOVL(498) D6656 D20160  ; 出料伺服Z轴#2腔取料位SV1, 出料伺服Z轴自动目标位置
LD TR0
AND W231.06  ; 出料伺服Z轴到#3腔取料位
MOVL(498) D6658 D20160  ; 出料伺服Z轴#3腔取料位SV1, 出料伺服Z轴自动目标位置
LD TR0
AND W231.12  ; 出料伺服Z轴到#4腔取料位
MOVL(498) D6660 D20160  ; 出料伺服Z轴#4腔取料位SV1, 出料伺服Z轴自动目标位置

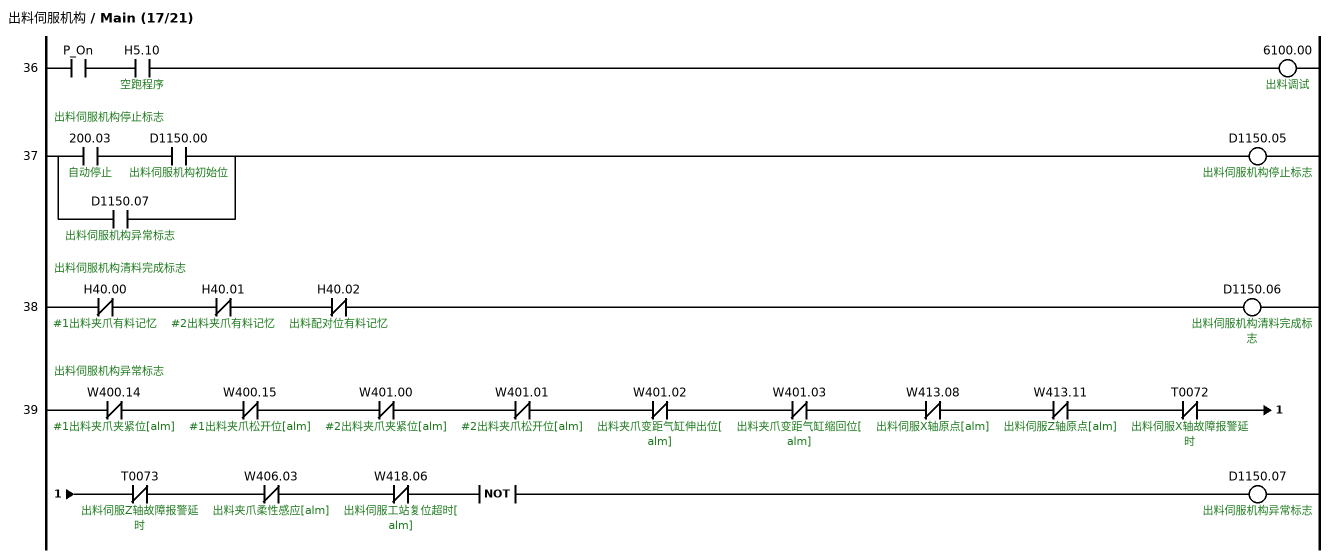
; rung 36
LD P_On
AND H5.10  ; 空跑程序
OUT 6100.00  ; 出料调试
; rung 37: 出料伺服机构停止标志
LD 200.03  ; 自动停止
AND D1150.00  ; 出料伺服机构初始位
OR D1150.07  ; 出料伺服机构异常标志
OUT D1150.05  ; 出料伺服机构停止标志
; rung 38: 出料伺服机构清料完成标志
LDNOT H40.00  ; #1出料夹爪有料记忆
ANDNOT H40.01  ; #2出料夹爪有料记忆
ANDNOT H40.02  ; 出料配对位有料记忆
OUT D1150.06  ; 出料伺服机构清料完成标志
; rung 39: 出料伺服机构异常标志
LDNOT W400.14  ; #1出料夹爪夹紧位[alm]
ANDNOT W400.15  ; #1出料夹爪松开位[alm]
ANDNOT W401.00  ; #2出料夹爪夹紧位[alm]
ANDNOT W401.01  ; #2出料夹爪松开位[alm]
ANDNOT W401.02  ; 出料夹爪变距气缸伸出位[alm]
ANDNOT W401.03  ; 出料夹爪变距气缸缩回位[alm]
ANDNOT W413.08  ; 出料伺服X轴原点[alm]
ANDNOT W413.11  ; 出料伺服Z轴原点[alm]
ANDNOT T0072  ; 出料伺服X轴故障报警延时
ANDNOT T0073  ; 出料伺服Z轴故障报警延时
ANDNOT W406.03  ; 出料夹爪柔性感应[alm]
ANDNOT W418.06  ; 出料伺服工站复位超时[alm]
NOT(520)
OUT D1150.07  ; 出料伺服机构异常标志

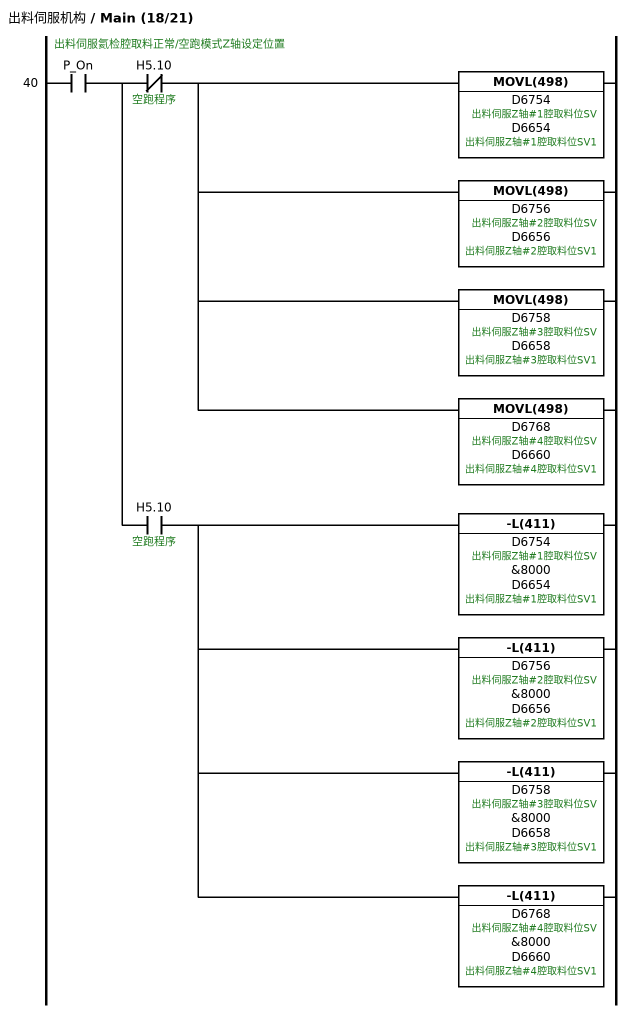
; rung 40: 出料伺服氦检腔取料正常/空跑模式Z轴设定位置
LD P_On
OUT TR0
ANDNOT H5.10  ; 空跑程序
MOVL(498) D6754 D6654  ; 出料伺服Z轴#1腔取料位SV, 出料伺服Z轴#1腔取料位SV1
MOVL(498) D6756 D6656  ; 出料伺服Z轴#2腔取料位SV, 出料伺服Z轴#2腔取料位SV1
MOVL(498) D6758 D6658  ; 出料伺服Z轴#3腔取料位SV, 出料伺服Z轴#3腔取料位SV1
MOVL(498) D6768 D6660  ; 出料伺服Z轴#4腔取料位SV, 出料伺服Z轴#4腔取料位SV1
LD TR0
AND H5.10  ; 空跑程序
-L(411) D6754 &8000 D6654  ; 出料伺服Z轴#1腔取料位SV, 出料伺服Z轴#1腔取料位SV1
-L(411) D6756 &8000 D6656  ; 出料伺服Z轴#2腔取料位SV, 出料伺服Z轴#2腔取料位SV1
-L(411) D6758 &8000 D6658  ; 出料伺服Z轴#3腔取料位SV, 出料伺服Z轴#3腔取料位SV1
-L(411) D6768 &8000 D6660  ; 出料伺服Z轴#4腔取料位SV, 出料伺服Z轴#4腔取料位SV1

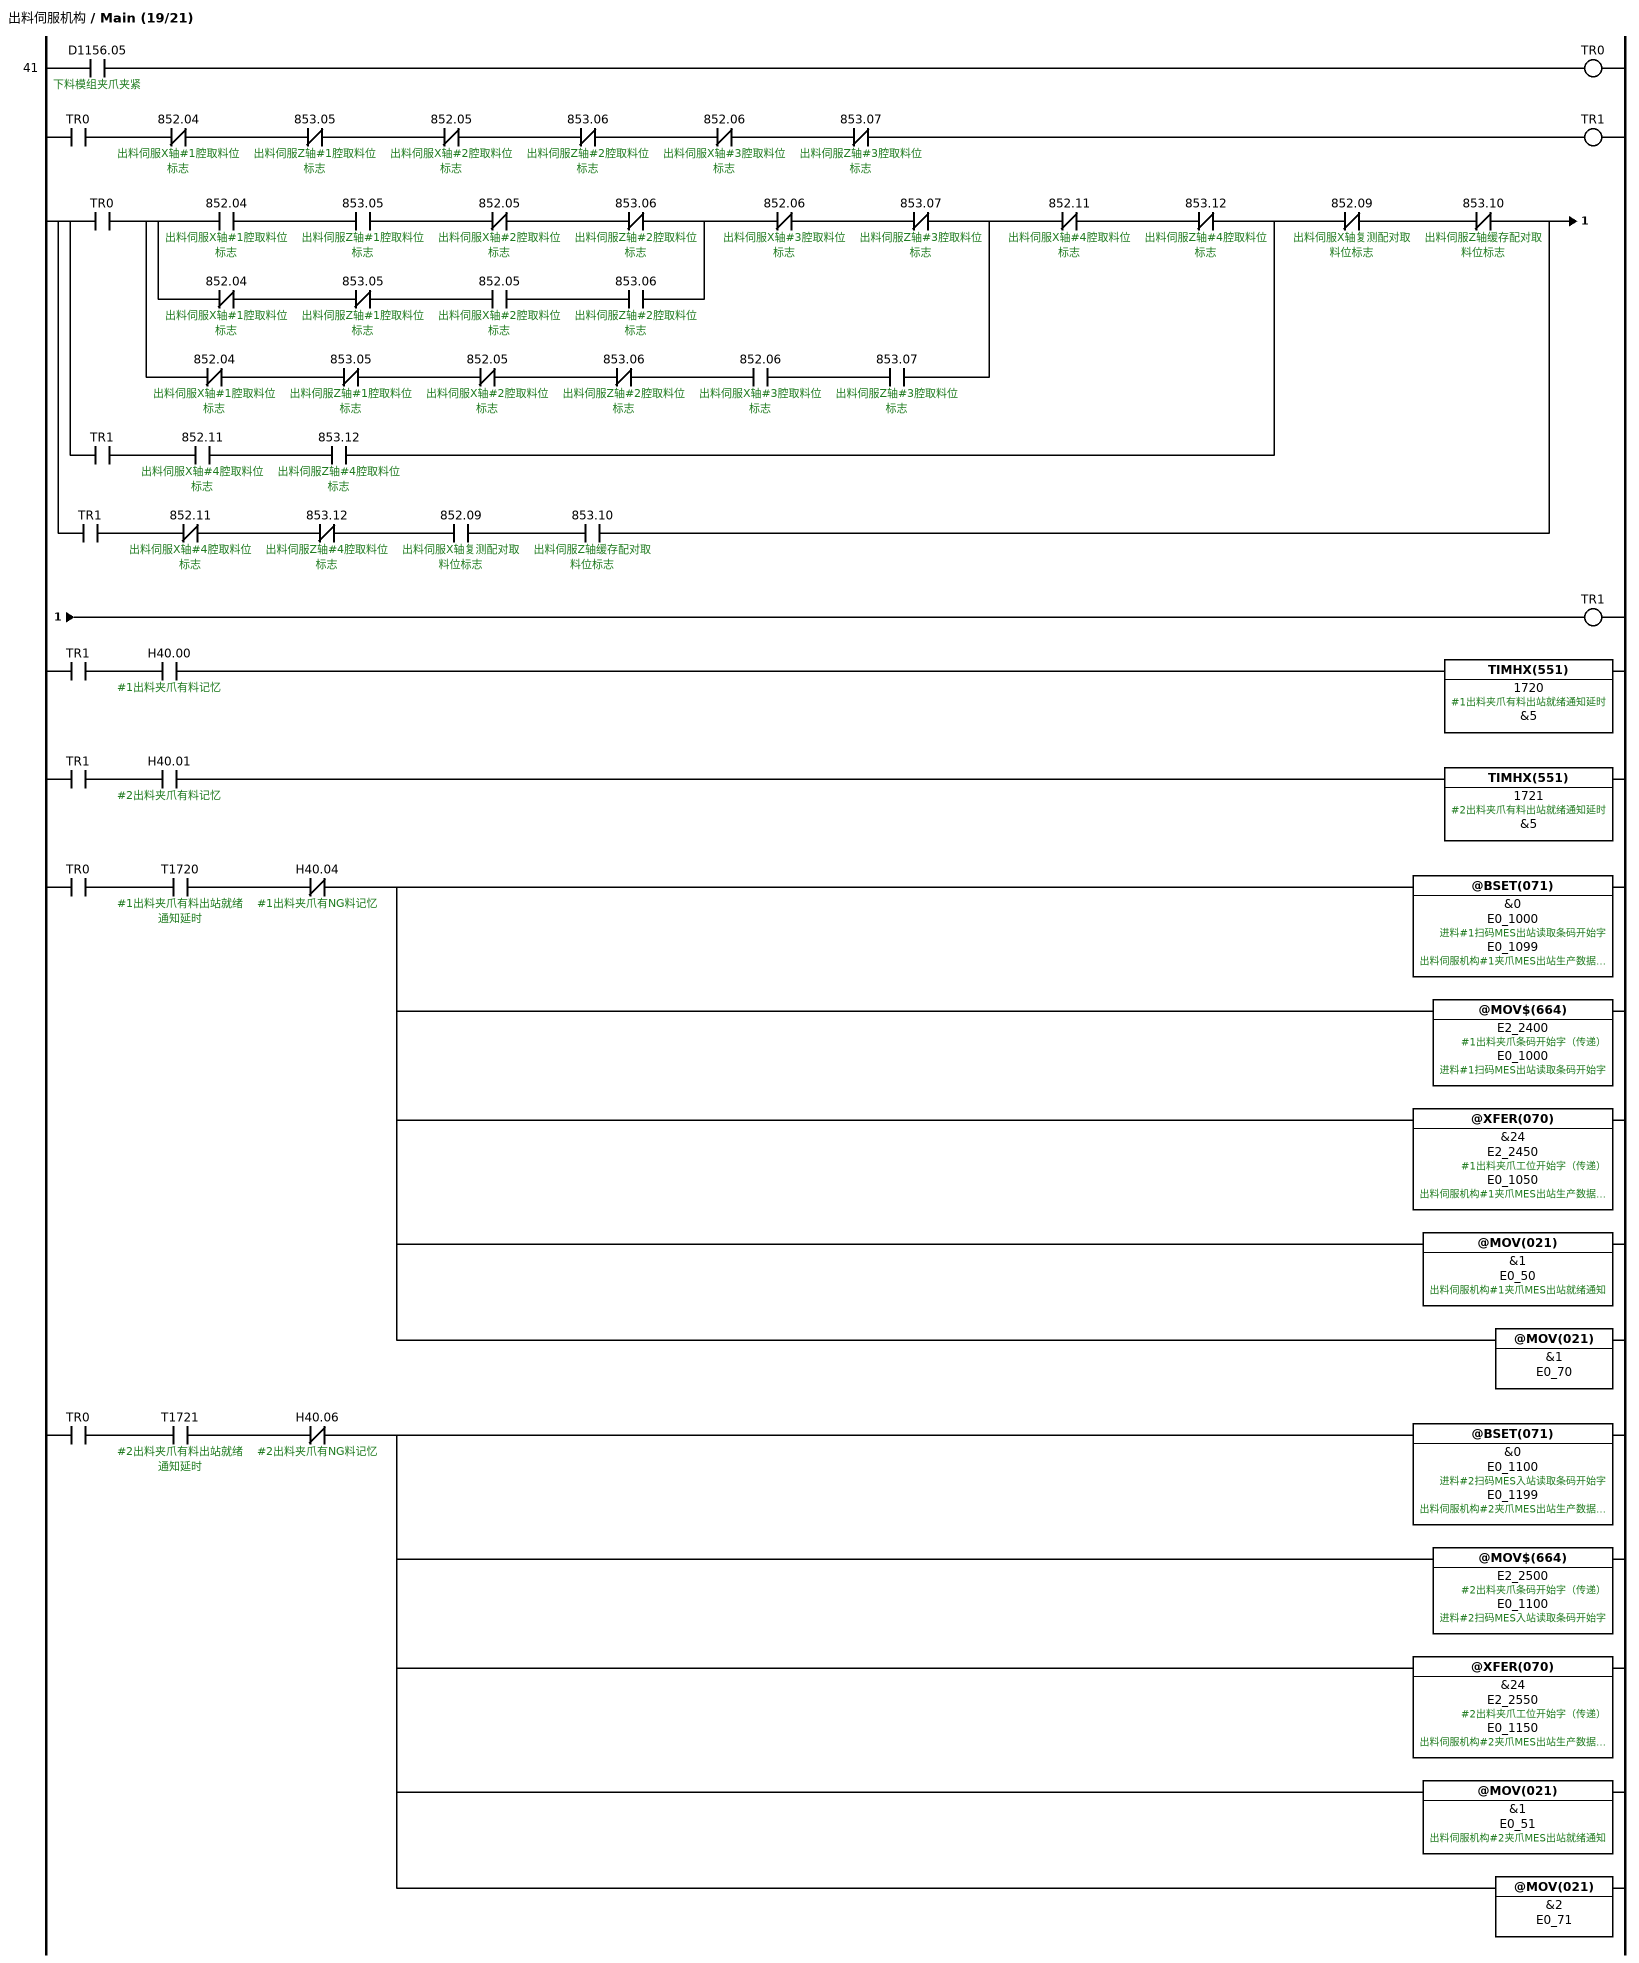
; rung 41
LD D1156.05  ; 下料模组夹爪夹紧
OUT TR0
LD 852.04  ; 出料伺服X轴#1腔取料位标志
AND 853.05  ; 出料伺服Z轴#1腔取料位标志
ANDNOT 852.05  ; 出料伺服X轴#2腔取料位标志
ANDNOT 853.06  ; 出料伺服Z轴#2腔取料位标志
LDNOT 852.04  ; 出料伺服X轴#1腔取料位标志
ANDNOT 853.05  ; 出料伺服Z轴#1腔取料位标志
AND 852.05  ; 出料伺服X轴#2腔取料位标志
AND 853.06  ; 出料伺服Z轴#2腔取料位标志
ORLD
ANDNOT 852.06  ; 出料伺服X轴#3腔取料位标志
ANDNOT 853.07  ; 出料伺服Z轴#3腔取料位标志
LDNOT 852.04  ; 出料伺服X轴#1腔取料位标志
ANDNOT 853.05  ; 出料伺服Z轴#1腔取料位标志
ANDNOT 852.05  ; 出料伺服X轴#2腔取料位标志
ANDNOT 853.06  ; 出料伺服Z轴#2腔取料位标志
AND 852.06  ; 出料伺服X轴#3腔取料位标志
AND 853.07  ; 出料伺服Z轴#3腔取料位标志
ORLD
ANDLD
ANDNOT 852.11  ; 出料伺服X轴#4腔取料位标志
ANDNOT 853.12  ; 出料伺服Z轴#4腔取料位标志
LD TR0
ANDNOT 852.04  ; 出料伺服X轴#1腔取料位标志
ANDNOT 853.05  ; 出料伺服Z轴#1腔取料位标志
ANDNOT 852.05  ; 出料伺服X轴#2腔取料位标志
ANDNOT 853.06  ; 出料伺服Z轴#2腔取料位标志
ANDNOT 852.06  ; 出料伺服X轴#3腔取料位标志
ANDNOT 853.07  ; 出料伺服Z轴#3腔取料位标志
OUT TR1
AND 852.11  ; 出料伺服X轴#4腔取料位标志
AND 853.12  ; 出料伺服Z轴#4腔取料位标志
ORLD
ANDNOT 852.09  ; 出料伺服X轴复测配对取料位标志
ANDNOT 853.10  ; 出料伺服Z轴缓存配对取料位标志
LD TR1
ANDNOT 852.11  ; 出料伺服X轴#4腔取料位标志
ANDNOT 853.12  ; 出料伺服Z轴#4腔取料位标志
AND 852.09  ; 出料伺服X轴复测配对取料位标志
AND 853.10  ; 出料伺服Z轴缓存配对取料位标志
ORLD
OUT TR1
AND H40.00  ; #1出料夹爪有料记忆
TIMHX(551) 1720 &5  ; #1出料夹爪有料出站就绪通知延时
LD TR1
AND H40.01  ; #2出料夹爪有料记忆
TIMHX(551) 1721 &5  ; #2出料夹爪有料出站就绪通知延时
LD TR0
AND T1720  ; #1出料夹爪有料出站就绪通知延时
ANDNOT H40.04  ; #1出料夹爪有NG料记忆
@BSET(071) &0 E0_1000 E0_1099  ; 进料#1扫码MES出站读取条码开始字, 出料伺服机构#1夹爪MES出站生产数据结束字
@MOV$(664) E2_2400 E0_1000  ; #1出料夹爪条码开始字（传递）, 进料#1扫码MES出站读取条码开始字
@XFER(070) &24 E2_2450 E0_1050  ; #1出料夹爪工位开始字（传递）, 出料伺服机构#1夹爪MES出站生产数据开始字
@MOV(021) &1 E0_50  ; 出料伺服机构#1夹爪MES出站就绪通知
@MOV(021) &1 E0_70
LD TR0
AND T1721  ; #2出料夹爪有料出站就绪通知延时
ANDNOT H40.06  ; #2出料夹爪有NG料记忆
@BSET(071) &0 E0_1100 E0_1199  ; 进料#2扫码MES入站读取条码开始字, 出料伺服机构#2夹爪MES出站生产数据结束字
@MOV$(664) E2_2500 E0_1100  ; #2出料夹爪条码开始字（传递）, 进料#2扫码MES入站读取条码开始字
@XFER(070) &24 E2_2550 E0_1150  ; #2出料夹爪工位开始字（传递）, 出料伺服机构#2夹爪MES出站生产数据开始字
@MOV(021) &1 E0_51  ; 出料伺服机构#2夹爪MES出站就绪通知
@MOV(021) &2 E0_71

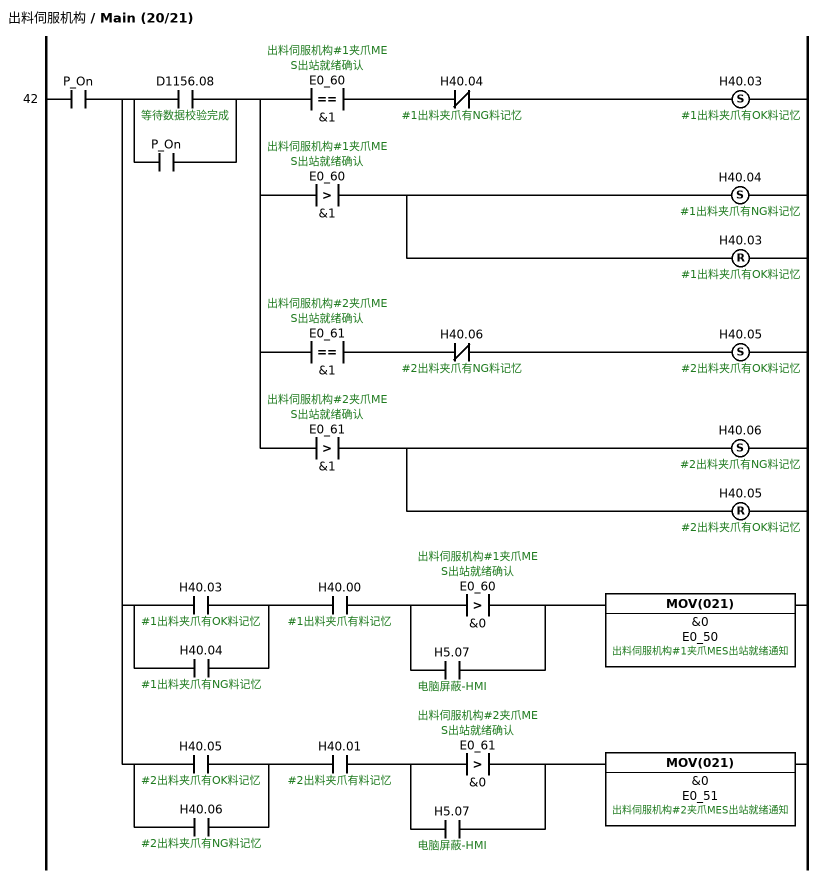
; rung 42
LD P_On
OUT TR0
LD D1156.08  ; 等待数据校验完成
OR P_On
ANDLD
OUT TR1
AND=(300) E0_60 &1  ; 出料伺服机构#1夹爪MES出站就绪确认
ANDNOT H40.04  ; #1出料夹爪有NG料记忆
SET H40.03  ; #1出料夹爪有OK料记忆
LD TR1
AND>(320) E0_60 &1  ; 出料伺服机构#1夹爪MES出站就绪确认
SET H40.04  ; #1出料夹爪有NG料记忆
RSET H40.03  ; #1出料夹爪有OK料记忆
LD TR1
AND=(300) E0_61 &1  ; 出料伺服机构#2夹爪MES出站就绪确认
ANDNOT H40.06  ; #2出料夹爪有NG料记忆
SET H40.05  ; #2出料夹爪有OK料记忆
LD TR1
AND>(320) E0_61 &1  ; 出料伺服机构#2夹爪MES出站就绪确认
SET H40.06  ; #2出料夹爪有NG料记忆
RSET H40.05  ; #2出料夹爪有OK料记忆
LD TR0
LD H40.03  ; #1出料夹爪有OK料记忆
OR H40.04  ; #1出料夹爪有NG料记忆
ANDLD
AND H40.00  ; #1出料夹爪有料记忆
LD>(320) E0_60 &0  ; 出料伺服机构#1夹爪MES出站就绪确认
OR H5.07  ; 电脑屏蔽-HMI
ANDLD
MOV(021) &0 E0_50  ; 出料伺服机构#1夹爪MES出站就绪通知
LD TR0
LD H40.05  ; #2出料夹爪有OK料记忆
OR H40.06  ; #2出料夹爪有NG料记忆
ANDLD
AND H40.01  ; #2出料夹爪有料记忆
LD>(320) E0_61 &0  ; 出料伺服机构#2夹爪MES出站就绪确认
OR H5.07  ; 电脑屏蔽-HMI
ANDLD
MOV(021) &0 E0_51  ; 出料伺服机构#2夹爪MES出站就绪通知

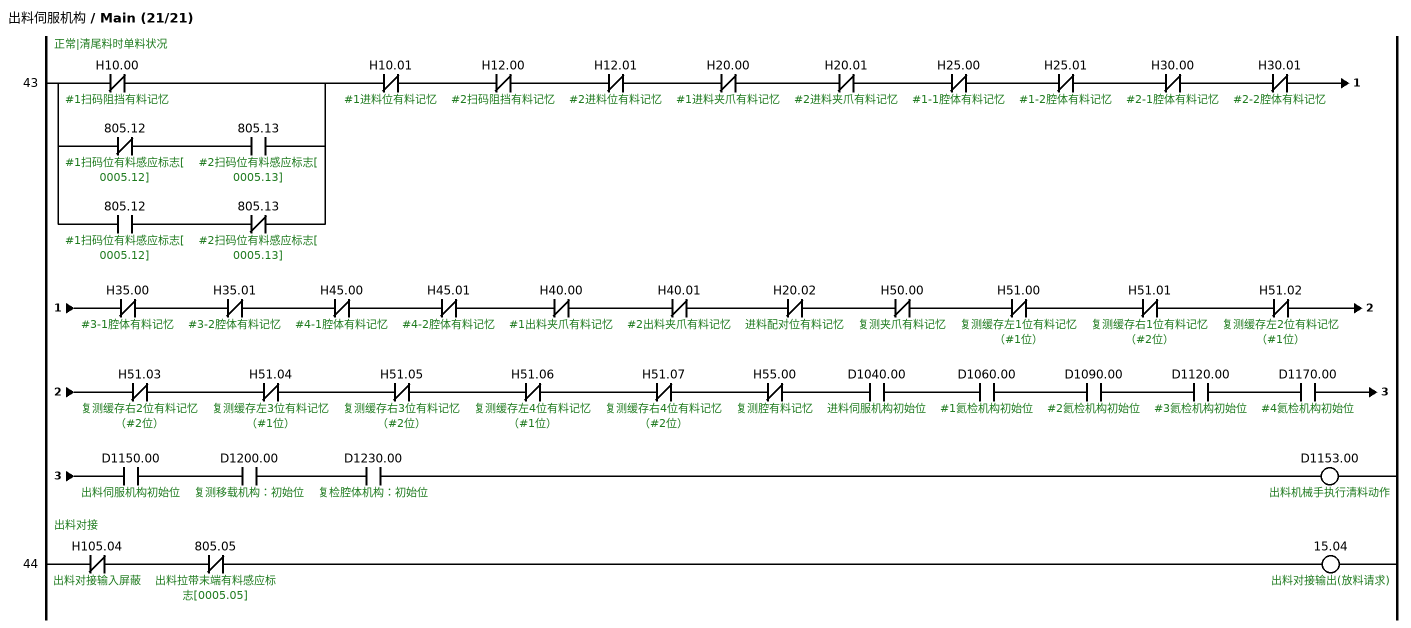
; rung 43: 正常|清尾料时单料状况
LDNOT H10.00  ; #1扫码阻挡有料记忆
LDNOT 805.12  ; #1扫码位有料感应标志[0005.12]
AND 805.13  ; #2扫码位有料感应标志[0005.13]
ORLD
LD 805.12  ; #1扫码位有料感应标志[0005.12]
ANDNOT 805.13  ; #2扫码位有料感应标志[0005.13]
ORLD
ANDNOT H10.01  ; #1进料位有料记忆
ANDNOT H12.00  ; #2扫码阻挡有料记忆
ANDNOT H12.01  ; #2进料位有料记忆
ANDNOT H20.00  ; #1进料夹爪有料记忆
ANDNOT H20.01  ; #2进料夹爪有料记忆
ANDNOT H25.00  ; #1-1腔体有料记忆
ANDNOT H25.01  ; #1-2腔体有料记忆
ANDNOT H30.00  ; #2-1腔体有料记忆
ANDNOT H30.01  ; #2-2腔体有料记忆
ANDNOT H35.00  ; #3-1腔体有料记忆
ANDNOT H35.01  ; #3-2腔体有料记忆
ANDNOT H45.00  ; #4-1腔体有料记忆
ANDNOT H45.01  ; #4-2腔体有料记忆
ANDNOT H40.00  ; #1出料夹爪有料记忆
ANDNOT H40.01  ; #2出料夹爪有料记忆
ANDNOT H20.02  ; 进料配对位有料记忆
ANDNOT H50.00  ; 复测夹爪有料记忆
ANDNOT H51.00  ; 复测缓存左1位有料记忆（#1位）
ANDNOT H51.01  ; 复测缓存右1位有料记忆（#2位）
ANDNOT H51.02  ; 复测缓存左2位有料记忆（#1位）
ANDNOT H51.03  ; 复测缓存右2位有料记忆（#2位）
ANDNOT H51.04  ; 复测缓存左3位有料记忆（#1位）
ANDNOT H51.05  ; 复测缓存右3位有料记忆（#2位）
ANDNOT H51.06  ; 复测缓存左4位有料记忆（#1位）
ANDNOT H51.07  ; 复测缓存右4位有料记忆（#2位）
ANDNOT H55.00  ; 复测腔有料记忆
AND D1040.00  ; 进料伺服机构初始位
AND D1060.00  ; #1氦检机构初始位
AND D1090.00  ; #2氦检机构初始位
AND D1120.00  ; #3氦检机构初始位
AND D1170.00  ; #4氦检机构初始位
AND D1150.00  ; 出料伺服机构初始位
AND D1200.00  ; 复测移载机构：初始位
AND D1230.00  ; 复检腔体机构：初始位
OUT D1153.00  ; 出料机械手执行清料动作
; rung 44: 出料对接
LDNOT H105.04  ; 出料对接输入屏蔽
ANDNOT 805.05  ; 出料拉带末端有料感应标志[0005.05]
OUT 15.04  ; 出料对接输出(放料请求)

### Section 出料伺服手动

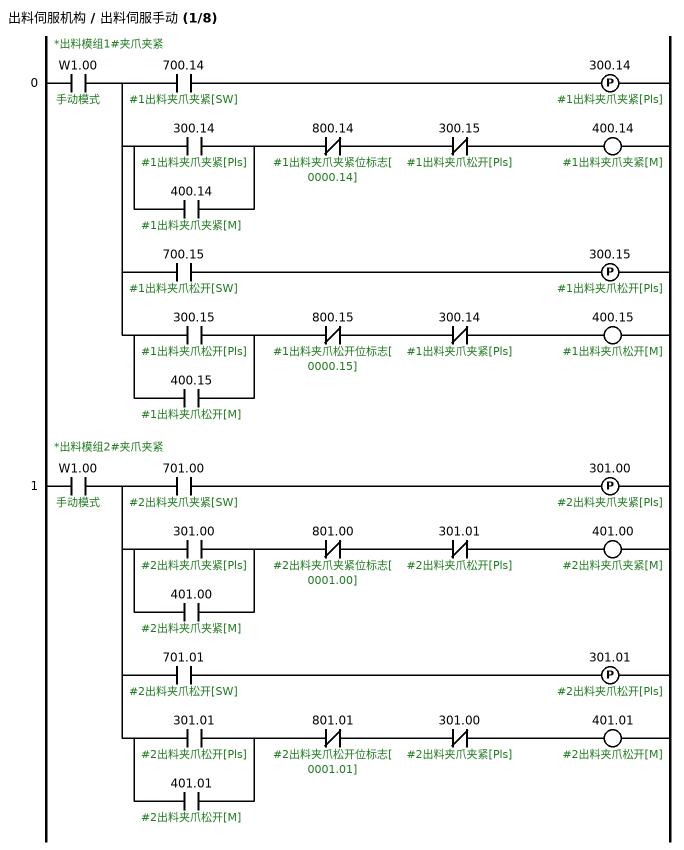
; rung 0: *出料模组1#夹爪夹紧
LD W1.00  ; 手动模式
OUT TR0
AND 700.14  ; #1出料夹爪夹紧[SW]
DIFU(013) 300.14  ; #1出料夹爪夹紧[Pls]
LD TR0
LD 300.14  ; #1出料夹爪夹紧[Pls]
OR 400.14  ; #1出料夹爪夹紧[M]
ANDLD
ANDNOT 800.14  ; #1出料夹爪夹紧位标志[0000.14]
ANDNOT 300.15  ; #1出料夹爪松开[Pls]
OUT 400.14  ; #1出料夹爪夹紧[M]
LD TR0
AND 700.15  ; #1出料夹爪松开[SW]
DIFU(013) 300.15  ; #1出料夹爪松开[Pls]
LD TR0
LD 300.15  ; #1出料夹爪松开[Pls]
OR 400.15  ; #1出料夹爪松开[M]
ANDLD
ANDNOT 800.15  ; #1出料夹爪松开位标志[0000.15]
ANDNOT 300.14  ; #1出料夹爪夹紧[Pls]
OUT 400.15  ; #1出料夹爪松开[M]
; rung 1: *出料模组2#夹爪夹紧
LD W1.00  ; 手动模式
OUT TR0
AND 701.00  ; #2出料夹爪夹紧[SW]
DIFU(013) 301.00  ; #2出料夹爪夹紧[Pls]
LD TR0
LD 301.00  ; #2出料夹爪夹紧[Pls]
OR 401.00  ; #2出料夹爪夹紧[M]
ANDLD
ANDNOT 801.00  ; #2出料夹爪夹紧位标志[0001.00]
ANDNOT 301.01  ; #2出料夹爪松开[Pls]
OUT 401.00  ; #2出料夹爪夹紧[M]
LD TR0
AND 701.01  ; #2出料夹爪松开[SW]
DIFU(013) 301.01  ; #2出料夹爪松开[Pls]
LD TR0
LD 301.01  ; #2出料夹爪松开[Pls]
OR 401.01  ; #2出料夹爪松开[M]
ANDLD
ANDNOT 801.01  ; #2出料夹爪松开位标志[0001.01]
ANDNOT 301.00  ; #2出料夹爪夹紧[Pls]
OUT 401.01  ; #2出料夹爪松开[M]

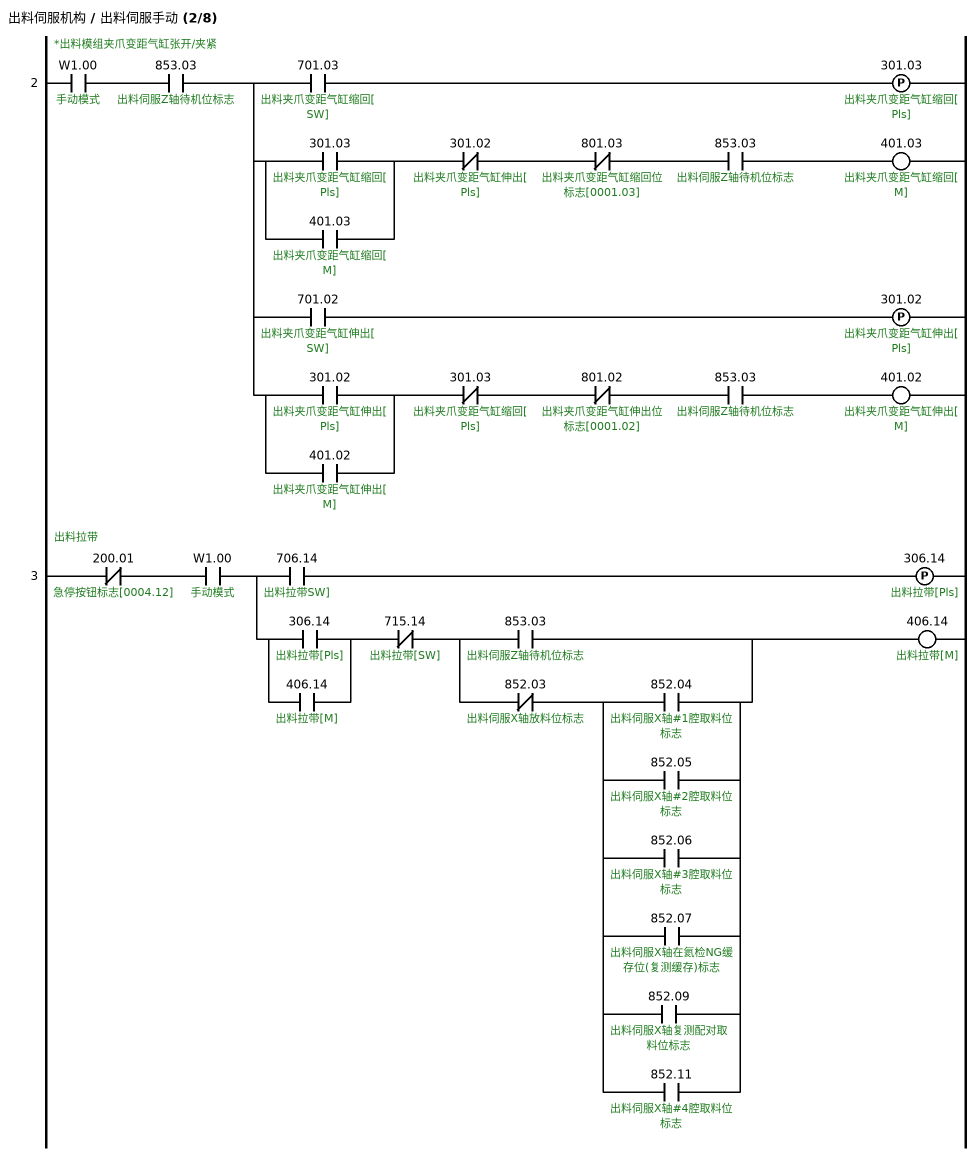
; rung 2: *出料模组夹爪变距气缸张开/夹紧
LD W1.00  ; 手动模式
AND 853.03  ; 出料伺服Z轴待机位标志
OUT TR0
AND 701.03  ; 出料夹爪变距气缸缩回[SW]
DIFU(013) 301.03  ; 出料夹爪变距气缸缩回[Pls]
LD TR0
LD 301.03  ; 出料夹爪变距气缸缩回[Pls]
OR 401.03  ; 出料夹爪变距气缸缩回[M]
ANDLD
ANDNOT 301.02  ; 出料夹爪变距气缸伸出[Pls]
ANDNOT 801.03  ; 出料夹爪变距气缸缩回位标志[0001.03]
AND 853.03  ; 出料伺服Z轴待机位标志
OUT 401.03  ; 出料夹爪变距气缸缩回[M]
LD TR0
AND 701.02  ; 出料夹爪变距气缸伸出[SW]
DIFU(013) 301.02  ; 出料夹爪变距气缸伸出[Pls]
LD TR0
LD 301.02  ; 出料夹爪变距气缸伸出[Pls]
OR 401.02  ; 出料夹爪变距气缸伸出[M]
ANDLD
ANDNOT 301.03  ; 出料夹爪变距气缸缩回[Pls]
ANDNOT 801.02  ; 出料夹爪变距气缸伸出位标志[0001.02]
AND 853.03  ; 出料伺服Z轴待机位标志
OUT 401.02  ; 出料夹爪变距气缸伸出[M]
; rung 3: 出料拉带
LDNOT 200.01  ; 急停按钮标志[0004.12]
AND W1.00  ; 手动模式
OUT TR0
AND 706.14  ; 出料拉带SW]
DIFU(013) 306.14  ; 出料拉带[Pls]
LD TR0
LD 306.14  ; 出料拉带[Pls]
OR 406.14  ; 出料拉带[M]
ANDLD
ANDNOT 715.14  ; 出料拉带[SW]
LD 853.03  ; 出料伺服Z轴待机位标志
LDNOT 852.03  ; 出料伺服X轴放料位标志
LD 852.04  ; 出料伺服X轴#1腔取料位标志
OR 852.05  ; 出料伺服X轴#2腔取料位标志
OR 852.06  ; 出料伺服X轴#3腔取料位标志
OR 852.07  ; 出料伺服X轴在氦检NG缓存位(复测缓存)标志
OR 852.09  ; 出料伺服X轴复测配对取料位标志
OR 852.11  ; 出料伺服X轴#4腔取料位标志
ANDLD
ORLD
ANDLD
OUT 406.14  ; 出料拉带[M]

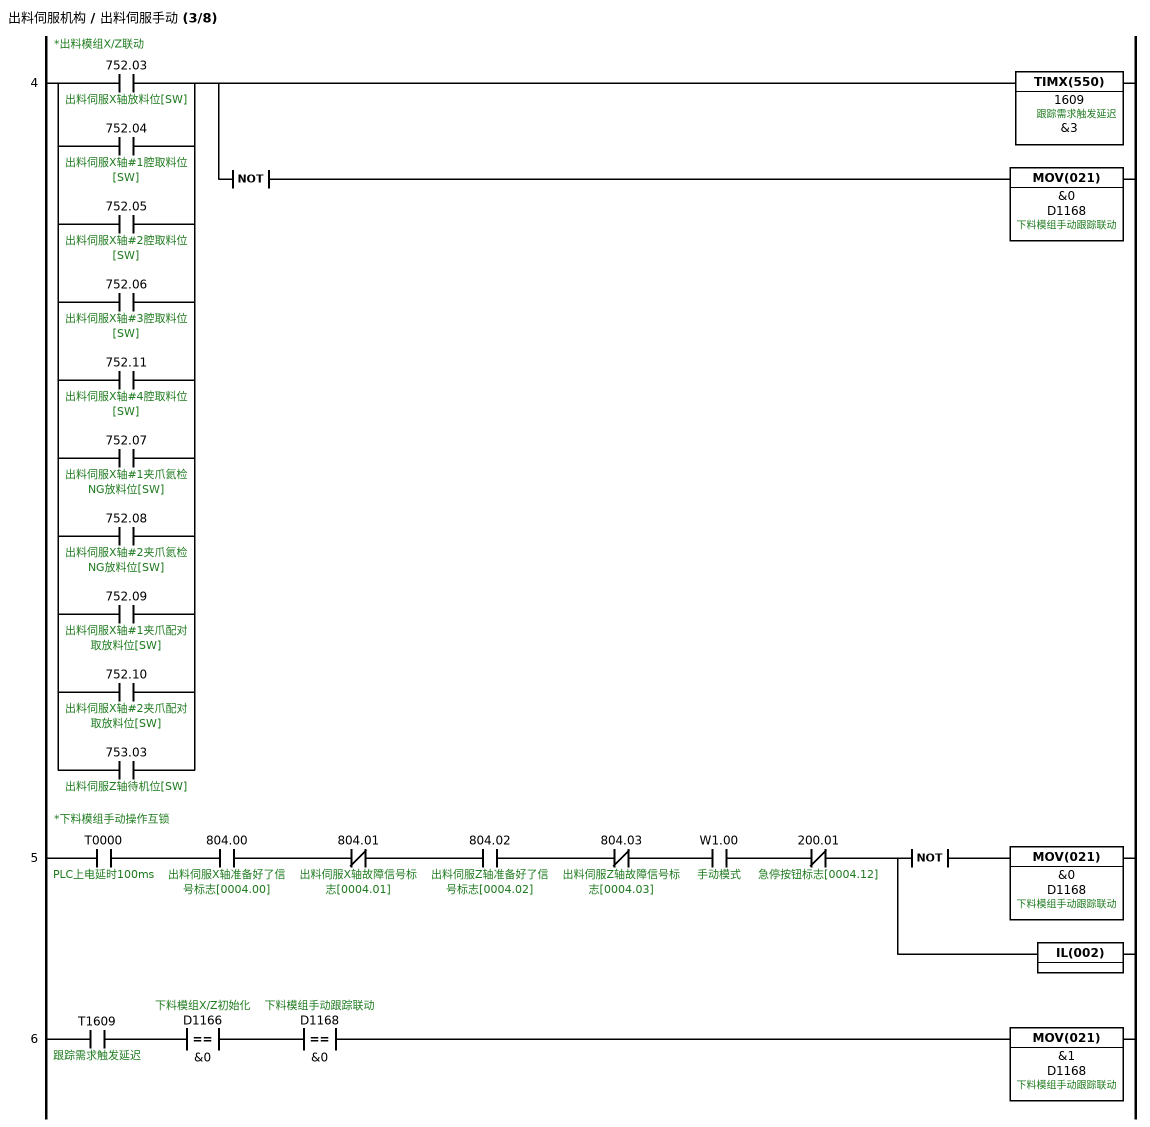
; rung 4: *出料模组X/Z联动
LD 752.03  ; 出料伺服X轴放料位[SW]
OR 752.04  ; 出料伺服X轴#1腔取料位[SW]
OR 752.05  ; 出料伺服X轴#2腔取料位[SW]
OR 752.06  ; 出料伺服X轴#3腔取料位[SW]
OR 752.11  ; 出料伺服X轴#4腔取料位[SW]
OR 752.07  ; 出料伺服X轴#1夹爪氦检NG放料位[SW]
OR 752.08  ; 出料伺服X轴#2夹爪氦检NG放料位[SW]
OR 752.09  ; 出料伺服X轴#1夹爪配对取放料位[SW]
OR 752.10  ; 出料伺服X轴#2夹爪配对取放料位[SW]
OR 753.03  ; 出料伺服Z轴待机位[SW]
TIMX(550) 1609 &3  ; 跟踪需求触发延迟
NOT(520)
MOV(021) &0 D1168  ; 下料模组手动跟踪联动
; rung 5: *下料模组手动操作互锁
LD T0000  ; PLC上电延时100ms
AND 804.00  ; 出料伺服X轴准备好了信号标志[0004.00]
ANDNOT 804.01  ; 出料伺服X轴故障信号标志[0004.01]
AND 804.02  ; 出料伺服Z轴准备好了信号标志[0004.02]
ANDNOT 804.03  ; 出料伺服Z轴故障信号标志[0004.03]
AND W1.00  ; 手动模式
ANDNOT 200.01  ; 急停按钮标志[0004.12]
OUT TR0
NOT(520)
MOV(021) &0 D1168  ; 下料模组手动跟踪联动
LD TR0
IL(002)
; rung 6
LD T1609  ; 跟踪需求触发延迟
AND=(300) D1166 &0  ; 下料模组X/Z初始化
AND=(300) D1168 &0  ; 下料模组手动跟踪联动
MOV(021) &1 D1168  ; 下料模组手动跟踪联动

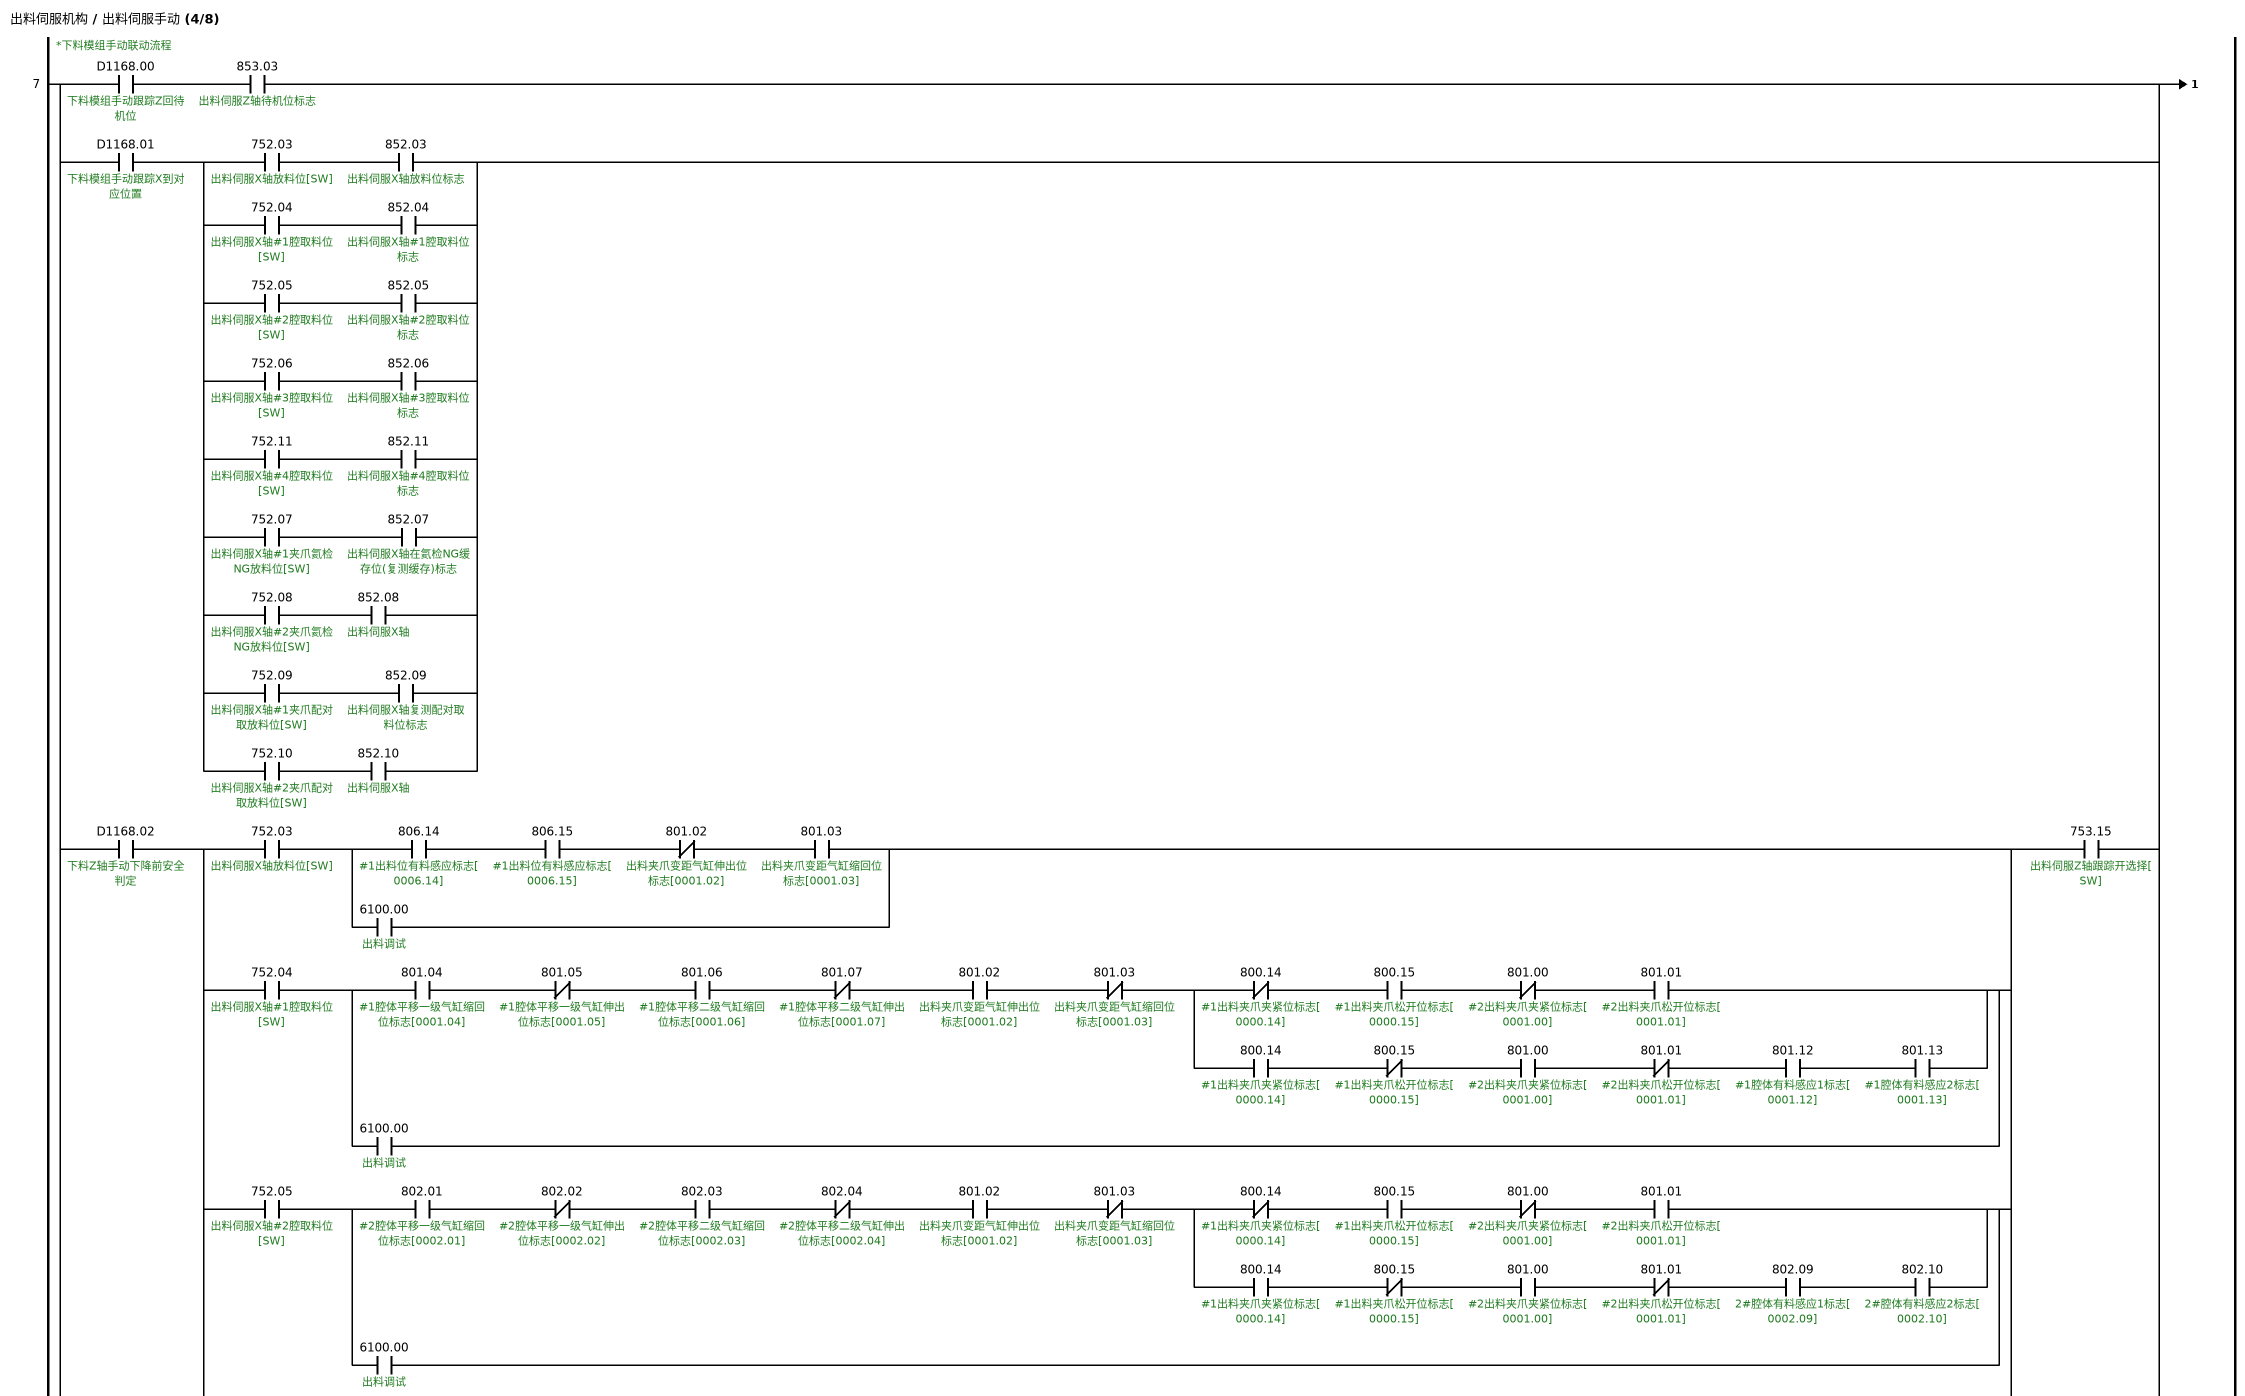

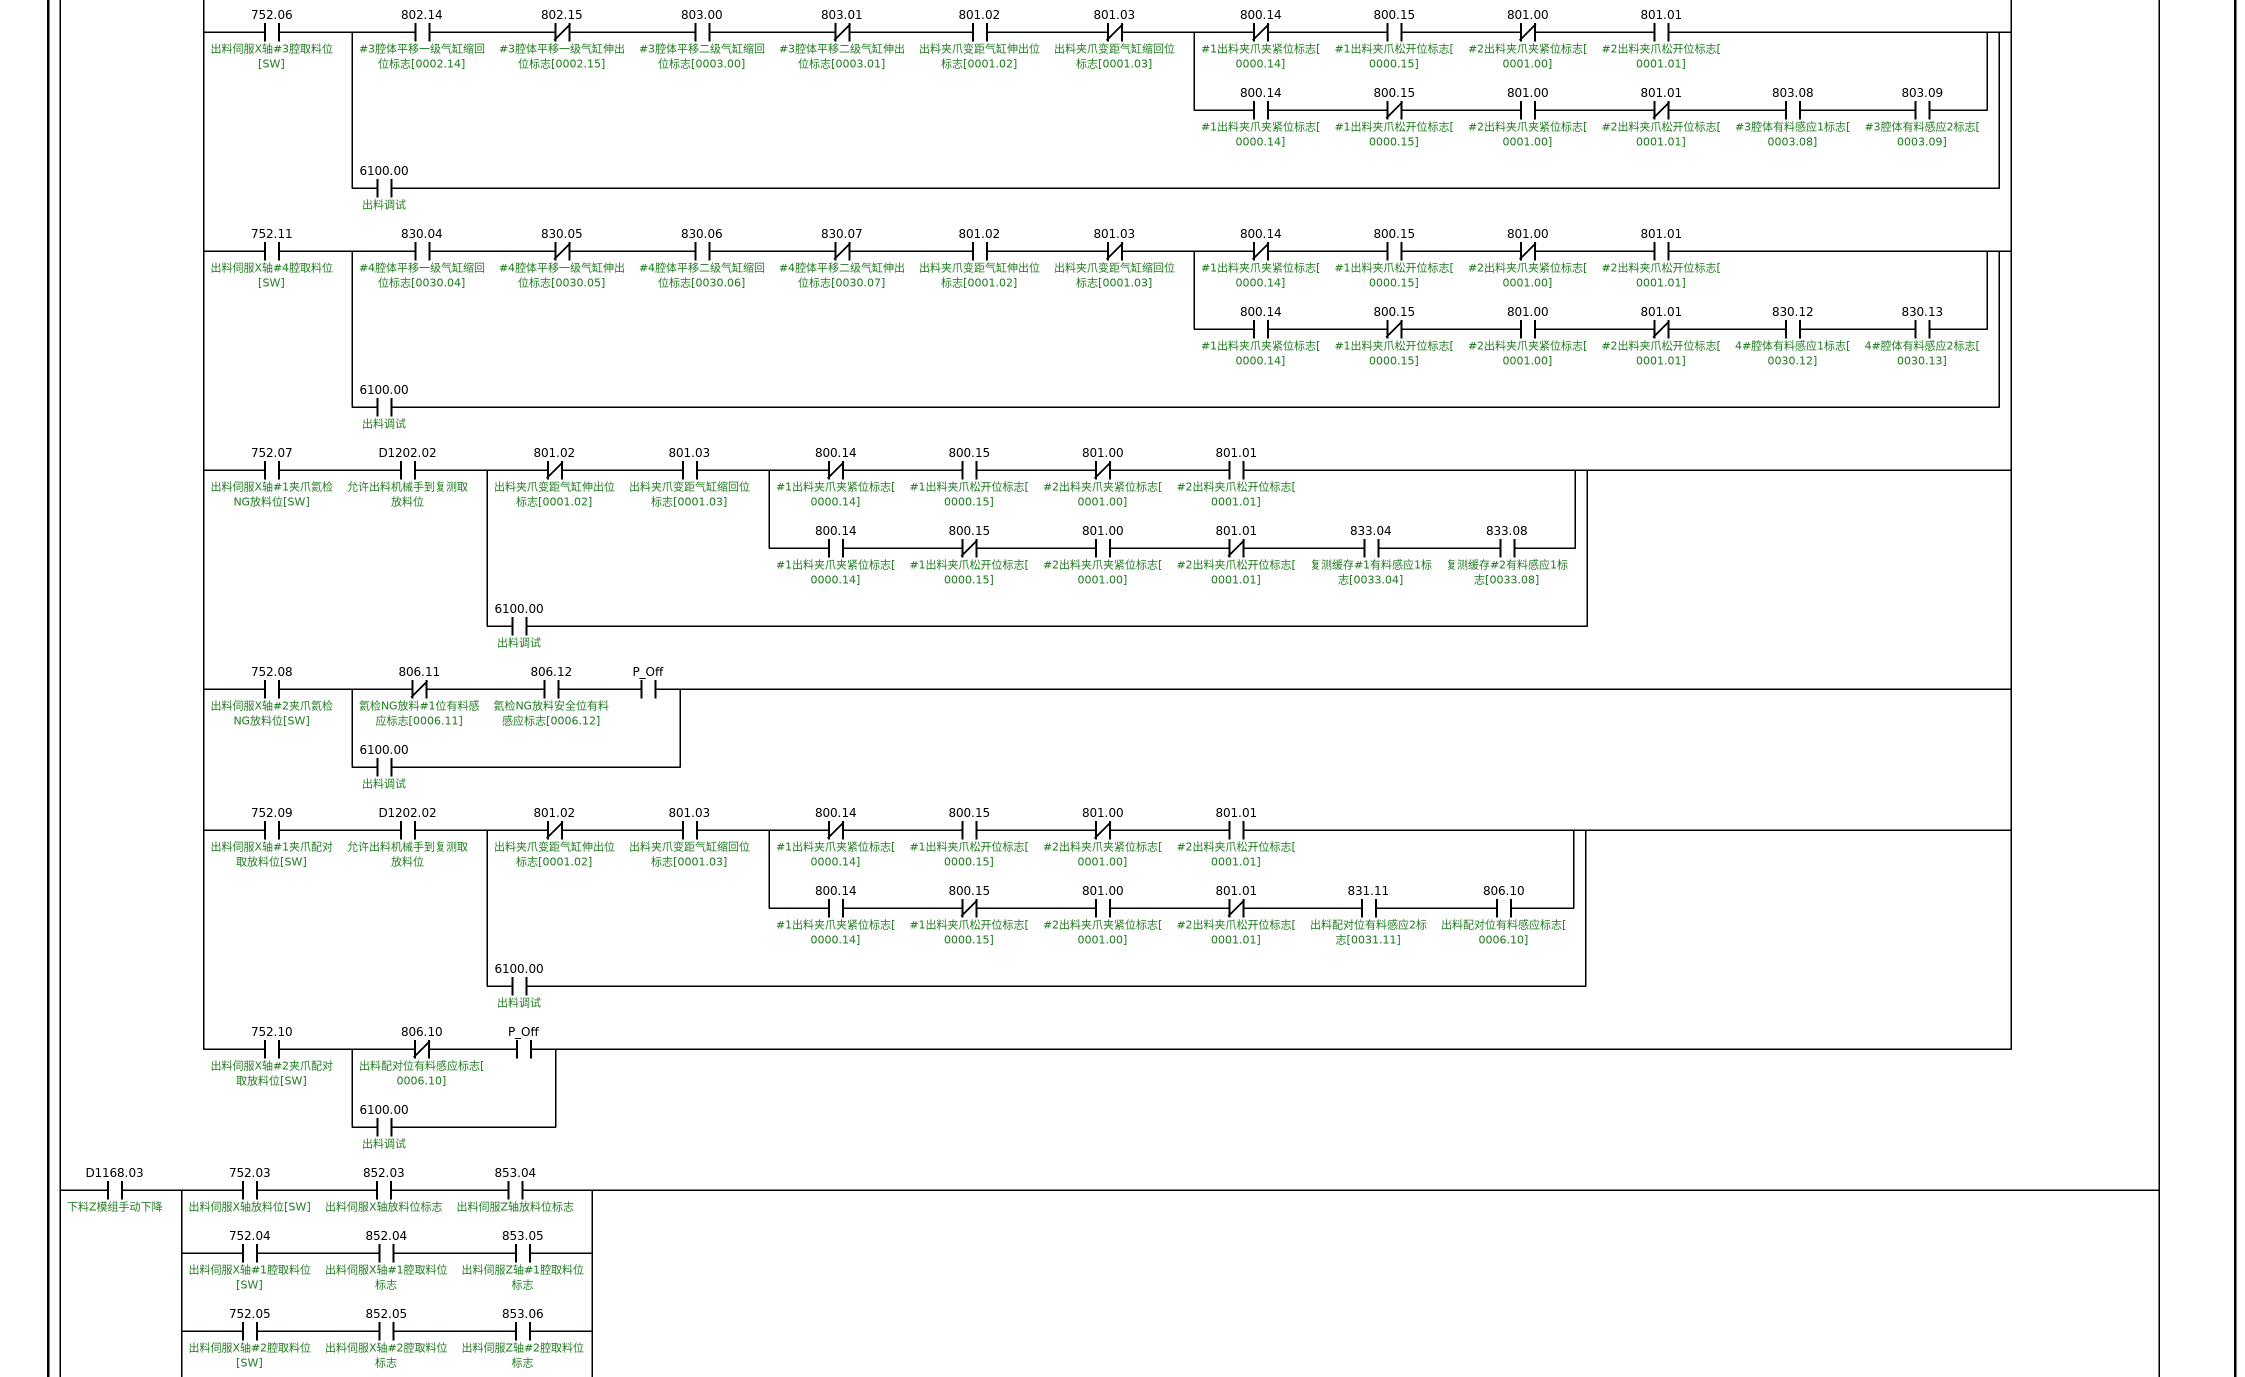

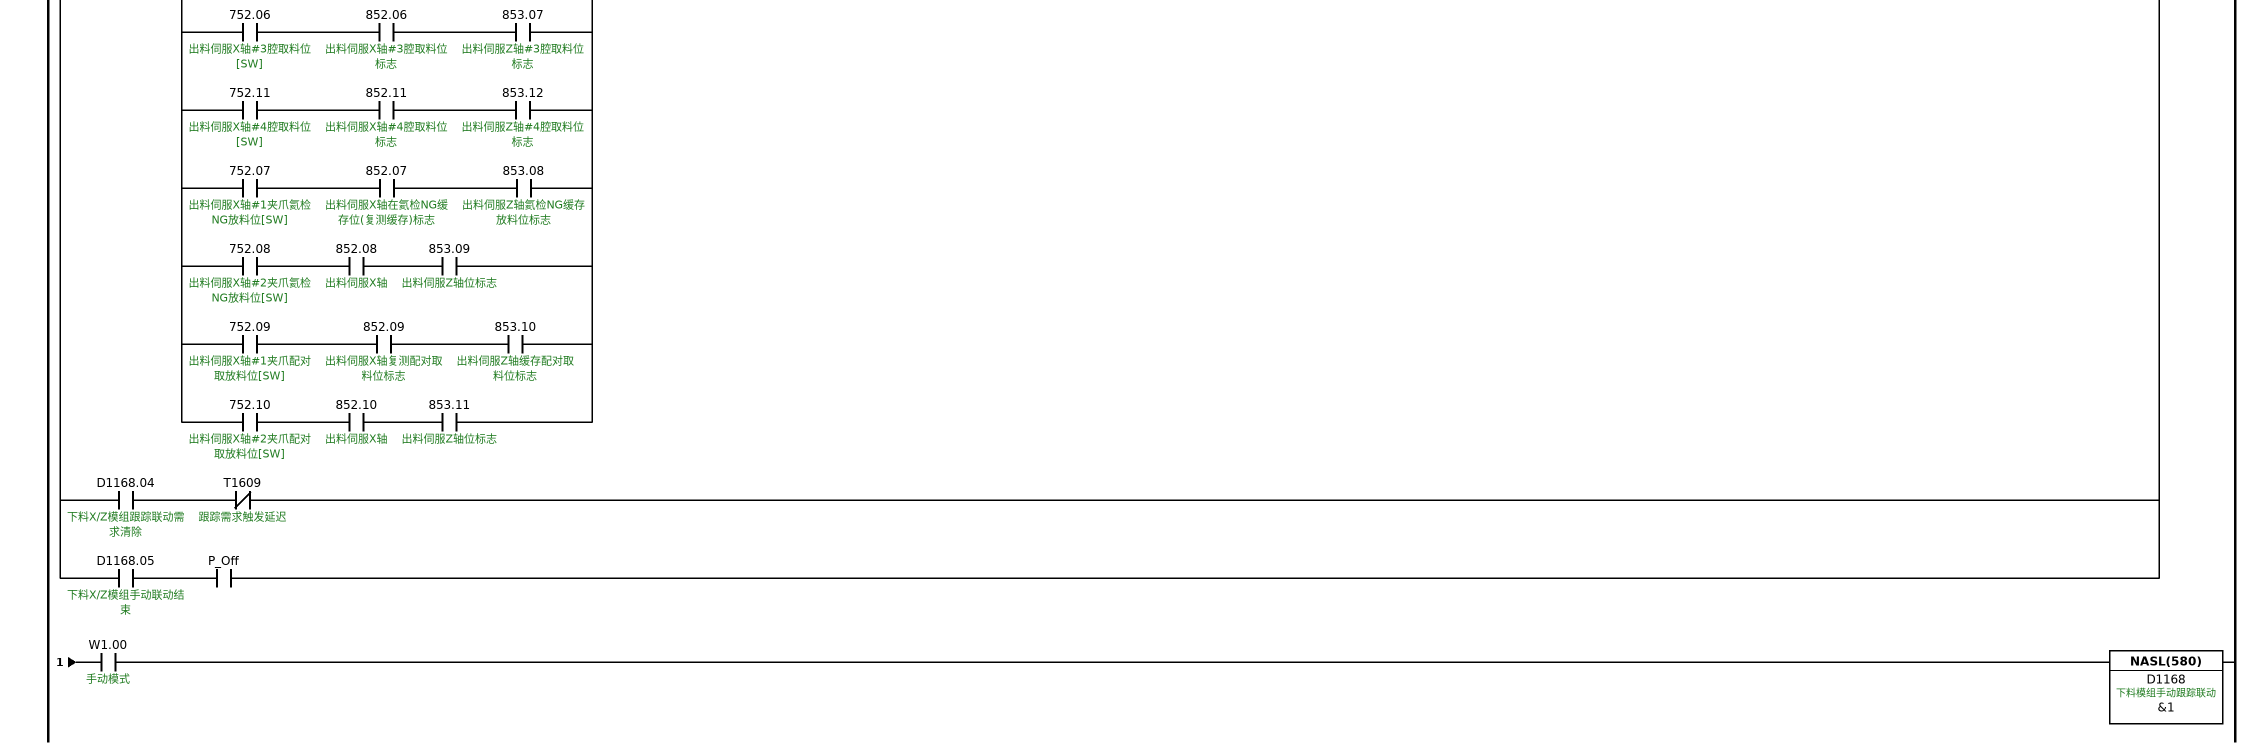
; rung 7: *下料模组手动联动流程
LD D1168.00  ; 下料模组手动跟踪Z回待机位
AND 853.03  ; 出料伺服Z轴待机位标志
LD D1168.01  ; 下料模组手动跟踪X到对应位置
LD 752.03  ; 出料伺服X轴放料位[SW]
AND 852.03  ; 出料伺服X轴放料位标志
LD 752.04  ; 出料伺服X轴#1腔取料位[SW]
AND 852.04  ; 出料伺服X轴#1腔取料位标志
ORLD
LD 752.05  ; 出料伺服X轴#2腔取料位[SW]
AND 852.05  ; 出料伺服X轴#2腔取料位标志
ORLD
LD 752.06  ; 出料伺服X轴#3腔取料位[SW]
AND 852.06  ; 出料伺服X轴#3腔取料位标志
ORLD
LD 752.11  ; 出料伺服X轴#4腔取料位[SW]
AND 852.11  ; 出料伺服X轴#4腔取料位标志
ORLD
LD 752.07  ; 出料伺服X轴#1夹爪氦检NG放料位[SW]
AND 852.07  ; 出料伺服X轴在氦检NG缓存位(复测缓存)标志
ORLD
LD 752.08  ; 出料伺服X轴#2夹爪氦检NG放料位[SW]
AND 852.08  ; 出料伺服X轴
ORLD
LD 752.09  ; 出料伺服X轴#1夹爪配对取放料位[SW]
AND 852.09  ; 出料伺服X轴复测配对取料位标志
ORLD
LD 752.10  ; 出料伺服X轴#2夹爪配对取放料位[SW]
AND 852.10  ; 出料伺服X轴
ORLD
ANDLD
ORLD
LD D1168.02  ; 下料Z轴手动下降前安全判定
LD 752.03  ; 出料伺服X轴放料位[SW]
LD 806.14  ; #1出料位有料感应标志[0006.14]
AND 806.15  ; #1出料位有料感应标志[0006.15]
ANDNOT 801.02  ; 出料夹爪变距气缸伸出位标志[0001.02]
AND 801.03  ; 出料夹爪变距气缸缩回位标志[0001.03]
OR 6100.00  ; 出料调试
ANDLD
LD 752.04  ; 出料伺服X轴#1腔取料位[SW]
LD 801.04  ; #1腔体平移一级气缸缩回位标志[0001.04]
ANDNOT 801.05  ; #1腔体平移一级气缸伸出位标志[0001.05]
AND 801.06  ; #1腔体平移二级气缸缩回位标志[0001.06]
ANDNOT 801.07  ; #1腔体平移二级气缸伸出位标志[0001.07]
AND 801.02  ; 出料夹爪变距气缸伸出位标志[0001.02]
ANDNOT 801.03  ; 出料夹爪变距气缸缩回位标志[0001.03]
LDNOT 800.14  ; #1出料夹爪夹紧位标志[0000.14]
AND 800.15  ; #1出料夹爪松开位标志[0000.15]
ANDNOT 801.00  ; #2出料夹爪夹紧位标志[0001.00]
AND 801.01  ; #2出料夹爪松开位标志[0001.01]
LD 800.14  ; #1出料夹爪夹紧位标志[0000.14]
ANDNOT 800.15  ; #1出料夹爪松开位标志[0000.15]
AND 801.00  ; #2出料夹爪夹紧位标志[0001.00]
ANDNOT 801.01  ; #2出料夹爪松开位标志[0001.01]
AND 801.12  ; #1腔体有料感应1标志[0001.12]
AND 801.13  ; #1腔体有料感应2标志[0001.13]
ORLD
ANDLD
OR 6100.00  ; 出料调试
ANDLD
ORLD
LD 752.05  ; 出料伺服X轴#2腔取料位[SW]
LD 802.01  ; #2腔体平移一级气缸缩回位标志[0002.01]
ANDNOT 802.02  ; #2腔体平移一级气缸伸出位标志[0002.02]
AND 802.03  ; #2腔体平移二级气缸缩回位标志[0002.03]
ANDNOT 802.04  ; #2腔体平移二级气缸伸出位标志[0002.04]
AND 801.02  ; 出料夹爪变距气缸伸出位标志[0001.02]
ANDNOT 801.03  ; 出料夹爪变距气缸缩回位标志[0001.03]
LDNOT 800.14  ; #1出料夹爪夹紧位标志[0000.14]
AND 800.15  ; #1出料夹爪松开位标志[0000.15]
ANDNOT 801.00  ; #2出料夹爪夹紧位标志[0001.00]
AND 801.01  ; #2出料夹爪松开位标志[0001.01]
LD 800.14  ; #1出料夹爪夹紧位标志[0000.14]
ANDNOT 800.15  ; #1出料夹爪松开位标志[0000.15]
AND 801.00  ; #2出料夹爪夹紧位标志[0001.00]
ANDNOT 801.01  ; #2出料夹爪松开位标志[0001.01]
AND 802.09  ; 2#腔体有料感应1标志[0002.09]
AND 802.10  ; 2#腔体有料感应2标志[0002.10]
ORLD
ANDLD
OR 6100.00  ; 出料调试
ANDLD
ORLD
LD 752.06  ; 出料伺服X轴#3腔取料位[SW]
LD 802.14  ; #3腔体平移一级气缸缩回位标志[0002.14]
ANDNOT 802.15  ; #3腔体平移一级气缸伸出位标志[0002.15]
AND 803.00  ; #3腔体平移二级气缸缩回位标志[0003.00]
ANDNOT 803.01  ; #3腔体平移二级气缸伸出位标志[0003.01]
AND 801.02  ; 出料夹爪变距气缸伸出位标志[0001.02]
ANDNOT 801.03  ; 出料夹爪变距气缸缩回位标志[0001.03]
LDNOT 800.14  ; #1出料夹爪夹紧位标志[0000.14]
AND 800.15  ; #1出料夹爪松开位标志[0000.15]
ANDNOT 801.00  ; #2出料夹爪夹紧位标志[0001.00]
AND 801.01  ; #2出料夹爪松开位标志[0001.01]
LD 800.14  ; #1出料夹爪夹紧位标志[0000.14]
ANDNOT 800.15  ; #1出料夹爪松开位标志[0000.15]
AND 801.00  ; #2出料夹爪夹紧位标志[0001.00]
ANDNOT 801.01  ; #2出料夹爪松开位标志[0001.01]
AND 803.08  ; #3腔体有料感应1标志[0003.08]
AND 803.09  ; #3腔体有料感应2标志[0003.09]
ORLD
ANDLD
OR 6100.00  ; 出料调试
ANDLD
ORLD
LD 752.11  ; 出料伺服X轴#4腔取料位[SW]
LD 830.04  ; #4腔体平移一级气缸缩回位标志[0030.04]
ANDNOT 830.05  ; #4腔体平移一级气缸伸出位标志[0030.05]
AND 830.06  ; #4腔体平移二级气缸缩回位标志[0030.06]
ANDNOT 830.07  ; #4腔体平移二级气缸伸出位标志[0030.07]
AND 801.02  ; 出料夹爪变距气缸伸出位标志[0001.02]
ANDNOT 801.03  ; 出料夹爪变距气缸缩回位标志[0001.03]
LDNOT 800.14  ; #1出料夹爪夹紧位标志[0000.14]
AND 800.15  ; #1出料夹爪松开位标志[0000.15]
ANDNOT 801.00  ; #2出料夹爪夹紧位标志[0001.00]
AND 801.01  ; #2出料夹爪松开位标志[0001.01]
LD 800.14  ; #1出料夹爪夹紧位标志[0000.14]
ANDNOT 800.15  ; #1出料夹爪松开位标志[0000.15]
AND 801.00  ; #2出料夹爪夹紧位标志[0001.00]
ANDNOT 801.01  ; #2出料夹爪松开位标志[0001.01]
AND 830.12  ; 4#腔体有料感应1标志[0030.12]
AND 830.13  ; 4#腔体有料感应2标志[0030.13]
ORLD
ANDLD
OR 6100.00  ; 出料调试
ANDLD
ORLD
LD 752.07  ; 出料伺服X轴#1夹爪氦检NG放料位[SW]
AND D1202.02  ; 允许出料机械手到复测取放料位
LDNOT 801.02  ; 出料夹爪变距气缸伸出位标志[0001.02]
AND 801.03  ; 出料夹爪变距气缸缩回位标志[0001.03]
LDNOT 800.14  ; #1出料夹爪夹紧位标志[0000.14]
AND 800.15  ; #1出料夹爪松开位标志[0000.15]
ANDNOT 801.00  ; #2出料夹爪夹紧位标志[0001.00]
AND 801.01  ; #2出料夹爪松开位标志[0001.01]
LD 800.14  ; #1出料夹爪夹紧位标志[0000.14]
ANDNOT 800.15  ; #1出料夹爪松开位标志[0000.15]
AND 801.00  ; #2出料夹爪夹紧位标志[0001.00]
ANDNOT 801.01  ; #2出料夹爪松开位标志[0001.01]
AND 833.04  ; 复测缓存#1有料感应1标志[0033.04]
AND 833.08  ; 复测缓存#2有料感应1标志[0033.08]
ORLD
ANDLD
OR 6100.00  ; 出料调试
ANDLD
ORLD
LD 752.08  ; 出料伺服X轴#2夹爪氦检NG放料位[SW]
LDNOT 806.11  ; 氦检NG放料#1位有料感应标志[0006.11]
AND 806.12  ; 氦检NG放料安全位有料感应标志[0006.12]
AND P_Off
OR 6100.00  ; 出料调试
ANDLD
ORLD
LD 752.09  ; 出料伺服X轴#1夹爪配对取放料位[SW]
AND D1202.02  ; 允许出料机械手到复测取放料位
LDNOT 801.02  ; 出料夹爪变距气缸伸出位标志[0001.02]
AND 801.03  ; 出料夹爪变距气缸缩回位标志[0001.03]
LDNOT 800.14  ; #1出料夹爪夹紧位标志[0000.14]
AND 800.15  ; #1出料夹爪松开位标志[0000.15]
ANDNOT 801.00  ; #2出料夹爪夹紧位标志[0001.00]
AND 801.01  ; #2出料夹爪松开位标志[0001.01]
LD 800.14  ; #1出料夹爪夹紧位标志[0000.14]
ANDNOT 800.15  ; #1出料夹爪松开位标志[0000.15]
AND 801.00  ; #2出料夹爪夹紧位标志[0001.00]
ANDNOT 801.01  ; #2出料夹爪松开位标志[0001.01]
AND 831.11  ; 出料配对位有料感应2标志[0031.11]
AND 806.10  ; 出料配对位有料感应标志[0006.10]
ORLD
ANDLD
OR 6100.00  ; 出料调试
ANDLD
ORLD
LD 752.10  ; 出料伺服X轴#2夹爪配对取放料位[SW]
LDNOT 806.10  ; 出料配对位有料感应标志[0006.10]
AND P_Off
OR 6100.00  ; 出料调试
ANDLD
ORLD
ANDLD
AND 753.15  ; 出料伺服Z轴跟踪开选择[SW]
ORLD
LD D1168.03  ; 下料Z模组手动下降
LD 752.03  ; 出料伺服X轴放料位[SW]
AND 852.03  ; 出料伺服X轴放料位标志
AND 853.04  ; 出料伺服Z轴放料位标志
LD 752.04  ; 出料伺服X轴#1腔取料位[SW]
AND 852.04  ; 出料伺服X轴#1腔取料位标志
AND 853.05  ; 出料伺服Z轴#1腔取料位标志
ORLD
LD 752.05  ; 出料伺服X轴#2腔取料位[SW]
AND 852.05  ; 出料伺服X轴#2腔取料位标志
AND 853.06  ; 出料伺服Z轴#2腔取料位标志
ORLD
LD 752.06  ; 出料伺服X轴#3腔取料位[SW]
AND 852.06  ; 出料伺服X轴#3腔取料位标志
AND 853.07  ; 出料伺服Z轴#3腔取料位标志
ORLD
LD 752.11  ; 出料伺服X轴#4腔取料位[SW]
AND 852.11  ; 出料伺服X轴#4腔取料位标志
AND 853.12  ; 出料伺服Z轴#4腔取料位标志
ORLD
LD 752.07  ; 出料伺服X轴#1夹爪氦检NG放料位[SW]
AND 852.07  ; 出料伺服X轴在氦检NG缓存位(复测缓存)标志
AND 853.08  ; 出料伺服Z轴氦检NG缓存放料位标志
ORLD
LD 752.08  ; 出料伺服X轴#2夹爪氦检NG放料位[SW]
AND 852.08  ; 出料伺服X轴
AND 853.09  ; 出料伺服Z轴位标志
ORLD
LD 752.09  ; 出料伺服X轴#1夹爪配对取放料位[SW]
AND 852.09  ; 出料伺服X轴复测配对取料位标志
AND 853.10  ; 出料伺服Z轴缓存配对取料位标志
ORLD
LD 752.10  ; 出料伺服X轴#2夹爪配对取放料位[SW]
AND 852.10  ; 出料伺服X轴
AND 853.11  ; 出料伺服Z轴位标志
ORLD
ANDLD
ORLD
LD D1168.04  ; 下料X/Z模组跟踪联动需求清除
ANDNOT T1609  ; 跟踪需求触发延迟
ORLD
LD D1168.05  ; 下料X/Z模组手动联动结束
AND P_Off
ORLD
AND W1.00  ; 手动模式
NASL(580) D1168 &1  ; 下料模组手动跟踪联动

